SPLINE
SPL {X  -134.737, Y  +296.229, Z    +0.000, E1   +47.890, E3 +135435.927}
SPL {X  -154.917, Y  +342.531, Z    +0.000, E1   +31.203, E3 +135454.495}
SPL {X  -159.440, Y  +369.246, Z    +0.000, E1   +13.458, E3 +135458.394}
SPL {X  -159.987, Y  +381.470, Z    +0.000, E1    +2.976, E3 +135458.993}
SPL {X  -159.990, Y  +384.500, Z    +0.000, E1    +0.000, E3 +135459.026}
SPL {X  -159.990, Y  +386.323, Z    +0.000, E1    -3.079, E3 +135459.048}
SPL {X  -159.990, Y  +390.285, Z    +0.000, E1   -11.315, E3 +135459.169}
SPL {X  -159.990, Y  +394.559, Z    +0.000, E1   -20.770, E3 +135459.431}
SPL {X  -159.990, Y  +399.334, Z    +0.000, E1   -30.876, E3 +135459.870}
SPL {X  -159.990, Y  +405.006, Z    +0.000, E1   -40.810, E3 +135460.588}
SPL {X  -159.990, Y  +415.193, Z    +0.000, E1   -52.724, E3 +135462.475}
SPL {X  -159.990, Y  +465.395, Z    +0.000, E1   -68.959, E3 +135477.563}
SPL {X  -159.990, Y  +657.157, Z    +0.000, E1   -72.499, E3 +135573.960}
SPL {X  -159.693, Y  +681.249, Z    +0.000, E1   -72.488, E3 +135590.354}
SPL {X  -157.599, Y  +699.059, Z    +0.000, E1   -72.249, E3 +135604.514}
SPL {X  -155.217, Y  +710.289, Z    +0.000, E1   -71.989, E3 +135614.530}
SPL {X  -152.611, Y  +719.527, Z    +0.000, E1   -71.702, E3 +135623.352}
SPL {X  -149.536, Y  +728.383, Z    +0.000, E1   -71.359, E3 +135632.331}
SPL {X  -146.250, Y  +736.367, Z    +0.000, E1   -70.965, E3 +135640.885}
SPL {X  -143.481, Y  +742.281, Z    +0.000, E1   -70.623, E3 +135647.480}
SPL {X  -140.071, Y  +748.811, Z    +0.000, E1   -70.193, E3 +135654.992}
SPL {X  -136.578, Y  +754.826, Z    +0.000, E1   -69.723, E3 +135662.122}
SPL {X  -132.176, Y  +761.646, Z    +0.000, E1   -69.128, E3 +135670.365}
SPL {X  -127.941, Y  +767.561, Z    +0.000, E1   -68.475, E3 +135677.673}
SPL {X  -124.983, Y  +771.380, Z    +0.000, E1   -68.003, E3 +135682.392}
SPL {X  -122.624, Y  +774.263, Z    +0.000, E1   -67.622, E3 +135685.915}
SPL {X   -84.435, Y  +807.395, Z    +0.000, E1   -55.948, E3 +135796.919}
ENDSPLINE

SPLINE
SPL {X  -119.703, Y  +777.650, Z    +0.000, E1   -51.831, E3 +135960.926}
SPL {X  -145.184, Y  +738.720, Z    +0.000, E1   -43.488, E3 +135987.484}
SPL {X  -156.175, Y  +706.232, Z    +0.000, E1   -28.819, E3 +135996.369}
SPL {X  -159.337, Y  +685.942, Z    +0.000, E1   -14.672, E3 +135998.920}
SPL {X  -159.962, Y  +674.468, Z    +0.000, E1    -4.846, E3 +135999.539}
SPL {X  -159.990, Y  +669.479, Z    +0.000, E1    +0.004, E3 +135999.613}
SPL {X  -159.990, Y  +667.035, Z    +0.000, E1    +4.539, E3 +135999.644}
SPL {X  -159.990, Y  +662.914, Z    +0.000, E1   +13.494, E3 +135999.782}
SPL {X  -159.990, Y  +658.254, Z    +0.000, E1   +24.153, E3 +136000.060}
SPL {X  -159.990, Y  +650.381, Z    +0.000, E1   +39.393, E3 +136000.912}
SPL {X  -159.990, Y  +638.701, Z    +0.000, E1   +53.953, E3 +136002.798}
SPL {X  -159.990, Y  +618.566, Z    +0.000, E1   +64.119, E3 +136008.306}
SPL {X  -159.990, Y  +582.261, Z    +0.000, E1   +69.343, E3 +136021.792}
SPL {X  -159.990, Y  +406.555, Z    +0.000, E1   +71.635, E3 +136118.038}
SPL {X  -159.990, Y  +385.723, Z    +0.000, E1   +71.610, E3 +136132.777}
SPL {X  -159.404, Y  +368.814, Z    +0.000, E1   +71.556, E3 +136145.306}
SPL {X  -157.440, Y  +354.048, Z    +0.000, E1   +71.342, E3 +136157.779}
SPL {X  -155.889, Y  +346.508, Z    +0.000, E1   +70.461, E3 +136171.327}
SPL {X  -154.332, Y  +340.328, Z    +0.000, E1   +70.024, E3 +136179.555}
SPL {X  -150.579, Y  +328.438, Z    +0.000, E1   +70.374, E3 +136185.274}
SPL {X  -146.933, Y  +319.195, Z    +0.000, E1   +70.230, E3 +136192.965}
SPL {X  -143.573, Y  +311.906, Z    +0.000, E1   +69.806, E3 +136201.275}
SPL {X  -139.693, Y  +304.508, Z    +0.000, E1   +69.301, E3 +136210.003}
SPL {X  -135.622, Y  +297.627, Z    +0.000, E1   +68.731, E3 +136218.411}
SPL {X  -131.165, Y  +290.889, Z    +0.000, E1   +68.094, E3 +136226.797}
SPL {X  -126.457, Y  +284.492, Z    +0.000, E1   +67.352, E3 +136234.882}
SPL {X  -123.432, Y  +280.710, Z    +0.000, E1   +66.830, E3 +136239.668}
SPL {X   -85.607, Y  +247.340, Z    +0.000, E1   +53.917, E3 +136381.389}
ENDSPLINE

SPLINE
SPL {X  -134.737, Y  +296.229, Z    +0.000, E1   +47.890, E3 +136524.162}
SPL {X  -154.917, Y  +342.531, Z    +0.000, E1   +31.203, E3 +136542.730}
SPL {X  -159.440, Y  +369.246, Z    +0.000, E1   +13.458, E3 +136546.629}
SPL {X  -159.987, Y  +381.470, Z    +0.000, E1    +2.976, E3 +136547.228}
SPL {X  -159.990, Y  +384.500, Z    +0.000, E1    +0.000, E3 +136547.261}
SPL {X  -159.990, Y  +386.323, Z    +0.000, E1    -3.079, E3 +136547.283}
SPL {X  -159.990, Y  +390.285, Z    +0.000, E1   -11.315, E3 +136547.404}
SPL {X  -159.990, Y  +394.559, Z    +0.000, E1   -20.770, E3 +136547.666}
SPL {X  -159.990, Y  +402.118, Z    +0.000, E1   -35.793, E3 +136548.457}
SPL {X  -159.990, Y  +415.193, Z    +0.000, E1   -52.724, E3 +136550.710}
SPL {X  -159.990, Y  +465.395, Z    +0.000, E1   -68.959, E3 +136565.799}
SPL {X  -159.990, Y  +652.170, Z    +0.000, E1   -72.485, E3 +136658.894}
SPL {X  -159.990, Y  +670.864, Z    +0.000, E1   -72.509, E3 +136671.342}
SPL {X  -159.251, Y  +686.856, Z    +0.000, E1   -72.412, E3 +136682.884}
SPL {X  -157.599, Y  +699.059, Z    +0.000, E1   -72.249, E3 +136692.749}
SPL {X  -155.217, Y  +710.289, Z    +0.000, E1   -71.989, E3 +136702.766}
SPL {X  -152.611, Y  +719.527, Z    +0.000, E1   -71.702, E3 +136711.587}
SPL {X  -149.536, Y  +728.383, Z    +0.000, E1   -71.359, E3 +136720.566}
SPL {X  -146.250, Y  +736.367, Z    +0.000, E1   -70.965, E3 +136729.120}
SPL {X  -143.481, Y  +742.281, Z    +0.000, E1   -70.623, E3 +136735.716}
SPL {X  -140.071, Y  +748.811, Z    +0.000, E1   -70.193, E3 +136743.227}
SPL {X  -136.578, Y  +754.826, Z    +0.000, E1   -69.723, E3 +136750.357}
SPL {X  -133.265, Y  +760.028, Z    +0.000, E1   -69.258, E3 +136756.658}
SPL {X  -129.890, Y  +764.909, Z    +0.000, E1   -68.775, E3 +136762.628}
SPL {X  -125.802, Y  +770.346, Z    +0.000, E1   -68.156, E3 +136769.328}
SPL {X  -122.624, Y  +774.263, Z    +0.000, E1   -67.622, E3 +136774.150}
SPL {X   -84.435, Y  +807.395, Z    +0.000, E1   -55.948, E3 +136885.155}
ENDSPLINE

SPLINE
SPL {X  -119.703, Y  +777.650, Z    +0.000, E1   -51.831, E3 +137049.161}
SPL {X  -145.184, Y  +738.720, Z    +0.000, E1   -43.488, E3 +137075.719}
SPL {X  -156.175, Y  +706.232, Z    +0.000, E1   -28.819, E3 +137084.604}
SPL {X  -159.337, Y  +685.942, Z    +0.000, E1   -14.672, E3 +137087.155}
SPL {X  -159.962, Y  +674.468, Z    +0.000, E1    -4.846, E3 +137087.774}
SPL {X  -159.990, Y  +669.479, Z    +0.000, E1    +0.004, E3 +137087.848}
SPL {X  -159.990, Y  +667.035, Z    +0.000, E1    +4.539, E3 +137087.879}
SPL {X  -159.990, Y  +662.914, Z    +0.000, E1   +13.494, E3 +137088.018}
SPL {X  -159.990, Y  +658.254, Z    +0.000, E1   +24.153, E3 +137088.295}
SPL {X  -159.990, Y  +652.944, Z    +0.000, E1   +35.122, E3 +137088.799}
SPL {X  -159.990, Y  +642.509, Z    +0.000, E1   +50.090, E3 +137090.371}
SPL {X  -159.990, Y  +618.566, Z    +0.000, E1   +64.119, E3 +137096.541}
SPL {X  -159.990, Y  +584.545, Z    +0.000, E1   +69.188, E3 +137109.076}
SPL {X  -159.990, Y  +578.002, Z    +0.000, E1   +69.607, E3 +137111.800}
SPL {X  -159.990, Y  +426.570, Z    +0.000, E1   +71.599, E3 +137192.290}
SPL {X  -159.990, Y  +405.946, Z    +0.000, E1   +71.630, E3 +137206.720}
SPL {X  -159.967, Y  +379.776, Z    +0.000, E1   +71.634, E3 +137225.167}
SPL {X  -158.535, Y  +360.970, Z    +0.000, E1   +71.460, E3 +137239.989}
SPL {X  -156.277, Y  +348.230, Z    +0.000, E1   +71.211, E3 +137251.332}
SPL {X  -155.351, Y  +344.251, Z    +0.000, E1   +70.004, E3 +137265.124}
SPL {X  -150.579, Y  +328.438, Z    +0.000, E1   +70.374, E3 +137273.509}
SPL {X  -146.933, Y  +319.195, Z    +0.000, E1   +70.230, E3 +137281.200}
SPL {X  -143.573, Y  +311.906, Z    +0.000, E1   +69.806, E3 +137289.510}
SPL {X  -139.693, Y  +304.508, Z    +0.000, E1   +69.301, E3 +137298.239}
SPL {X  -135.622, Y  +297.627, Z    +0.000, E1   +68.731, E3 +137306.647}
SPL {X  -131.165, Y  +290.889, Z    +0.000, E1   +68.094, E3 +137315.032}
SPL {X  -126.457, Y  +284.492, Z    +0.000, E1   +67.352, E3 +137323.118}
SPL {X  -123.432, Y  +280.710, Z    +0.000, E1   +66.830, E3 +137327.903}
SPL {X   -85.607, Y  +247.340, Z    +0.000, E1   +53.917, E3 +137469.625}
ENDSPLINE

SPLINE
SPL {X  -134.737, Y  +296.229, Z    +0.000, E1   +47.890, E3 +137612.398}
SPL {X  -154.917, Y  +342.531, Z    +0.000, E1   +31.203, E3 +137630.965}
SPL {X  -159.440, Y  +369.246, Z    +0.000, E1   +13.458, E3 +137634.864}
SPL {X  -159.957, Y  +379.264, Z    +0.000, E1    +4.909, E3 +137635.421}
SPL {X  -159.990, Y  +384.670, Z    +0.000, E1    -0.079, E3 +137635.498}
SPL {X  -159.990, Y  +389.248, Z    +0.000, E1    -8.879, E3 +137635.602}
SPL {X  -159.990, Y  +394.559, Z    +0.000, E1   -20.770, E3 +137635.901}
SPL {X  -159.990, Y  +402.118, Z    +0.000, E1   -35.793, E3 +137636.693}
SPL {X  -159.990, Y  +415.193, Z    +0.000, E1   -52.724, E3 +137638.945}
SPL {X  -159.990, Y  +465.395, Z    +0.000, E1   -68.959, E3 +137654.034}
SPL {X  -159.990, Y  +657.157, Z    +0.000, E1   -72.499, E3 +137750.431}
SPL {X  -159.947, Y  +675.227, Z    +0.000, E1   -72.487, E3 +137762.591}
SPL {X  -159.251, Y  +686.856, Z    +0.000, E1   -72.412, E3 +137771.119}
SPL {X  -157.599, Y  +699.059, Z    +0.000, E1   -72.249, E3 +137780.984}
SPL {X  -155.217, Y  +710.289, Z    +0.000, E1   -71.989, E3 +137791.001}
SPL {X  -152.611, Y  +719.527, Z    +0.000, E1   -71.702, E3 +137799.822}
SPL {X  -149.536, Y  +728.383, Z    +0.000, E1   -71.359, E3 +137808.801}
SPL {X  -146.250, Y  +736.367, Z    +0.000, E1   -70.965, E3 +137817.356}
SPL {X  -143.481, Y  +742.281, Z    +0.000, E1   -70.623, E3 +137823.951}
SPL {X  -140.071, Y  +748.811, Z    +0.000, E1   -70.193, E3 +137831.463}
SPL {X  -136.578, Y  +754.826, Z    +0.000, E1   -69.723, E3 +137838.592}
SPL {X  -133.265, Y  +760.028, Z    +0.000, E1   -69.258, E3 +137844.893}
SPL {X  -129.890, Y  +764.909, Z    +0.000, E1   -68.775, E3 +137850.864}
SPL {X  -125.802, Y  +770.346, Z    +0.000, E1   -68.156, E3 +137857.563}
SPL {X  -122.624, Y  +774.263, Z    +0.000, E1   -67.622, E3 +137862.386}
SPL {X   -84.435, Y  +807.395, Z    +0.000, E1   -55.948, E3 +137973.390}
ENDSPLINE

SPLINE
SPL {X  -119.703, Y  +777.650, Z    +0.000, E1   -51.831, E3 +138137.397}
SPL {X  -145.184, Y  +738.720, Z    +0.000, E1   -43.488, E3 +138163.955}
SPL {X  -154.467, Y  +713.173, Z    +0.000, E1   -32.658, E3 +138171.550}
SPL {X  -157.530, Y  +699.446, Z    +0.000, E1   -24.482, E3 +138173.966}
SPL {X  -159.337, Y  +685.942, Z    +0.000, E1   -14.672, E3 +138175.391}
SPL {X  -159.962, Y  +674.468, Z    +0.000, E1    -4.846, E3 +138176.009}
SPL {X  -159.990, Y  +669.479, Z    +0.000, E1    +0.004, E3 +138176.083}
SPL {X  -159.990, Y  +667.035, Z    +0.000, E1    +4.539, E3 +138176.114}
SPL {X  -159.990, Y  +662.914, Z    +0.000, E1   +13.494, E3 +138176.253}
SPL {X  -159.990, Y  +658.254, Z    +0.000, E1   +24.153, E3 +138176.531}
SPL {X  -159.990, Y  +652.944, Z    +0.000, E1   +35.122, E3 +138177.034}
SPL {X  -159.990, Y  +642.509, Z    +0.000, E1   +50.090, E3 +138178.606}
SPL {X  -159.990, Y  +618.566, Z    +0.000, E1   +64.119, E3 +138184.777}
SPL {X  -159.990, Y  +582.261, Z    +0.000, E1   +69.343, E3 +138198.262}
SPL {X  -159.990, Y  +406.555, Z    +0.000, E1   +71.635, E3 +138294.509}
SPL {X  -159.990, Y  +385.723, Z    +0.000, E1   +71.610, E3 +138309.247}
SPL {X  -159.700, Y  +372.863, Z    +0.000, E1   +71.570, E3 +138318.653}
SPL {X  -158.535, Y  +360.970, Z    +0.000, E1   +71.460, E3 +138328.224}
SPL {X  -156.277, Y  +348.230, Z    +0.000, E1   +71.211, E3 +138339.567}
SPL {X  -155.351, Y  +344.251, Z    +0.000, E1   +70.004, E3 +138353.359}
SPL {X  -150.579, Y  +328.438, Z    +0.000, E1   +70.374, E3 +138361.744}
SPL {X  -146.933, Y  +319.195, Z    +0.000, E1   +70.230, E3 +138369.435}
SPL {X  -143.573, Y  +311.906, Z    +0.000, E1   +69.806, E3 +138377.746}
SPL {X  -140.547, Y  +306.057, Z    +0.000, E1   +69.399, E3 +138384.638}
SPL {X  -137.438, Y  +300.600, Z    +0.000, E1   +68.984, E3 +138391.232}
SPL {X  -133.397, Y  +294.172, Z    +0.000, E1   +68.416, E3 +138399.167}
SPL {X  -128.822, Y  +287.623, Z    +0.000, E1   +67.729, E3 +138407.391}
SPL {X  -124.502, Y  +282.021, Z    +0.000, E1   +67.035, E3 +138414.465}
SPL {X   -85.607, Y  +247.340, Z    +0.000, E1   +53.917, E3 +138557.860}
ENDSPLINE

SPLINE
SPL {X  -119.557, Y  +276.184, Z    +0.000, E1   +51.032, E3 +138681.397}
SPL {X  -138.294, Y  +302.054, Z    +0.000, E1   +46.576, E3 +138704.719}
SPL {X  -153.211, Y  +336.421, Z    +0.000, E1   +34.262, E3 +138717.841}
SPL {X  -158.240, Y  +358.900, Z    +0.000, E1   +21.089, E3 +138722.046}
SPL {X  -159.674, Y  +372.451, Z    +0.000, E1   +10.778, E3 +138723.342}
SPL {X  -159.987, Y  +381.470, Z    +0.000, E1    +2.976, E3 +138723.699}
SPL {X  -159.990, Y  +384.761, Z    +0.000, E1    -0.257, E3 +138723.734}
SPL {X  -159.990, Y  +389.248, Z    +0.000, E1    -8.879, E3 +138723.838}
SPL {X  -159.990, Y  +394.559, Z    +0.000, E1   -20.770, E3 +138724.137}
SPL {X  -159.990, Y  +402.118, Z    +0.000, E1   -35.793, E3 +138724.928}
SPL {X  -159.990, Y  +415.193, Z    +0.000, E1   -52.724, E3 +138727.181}
SPL {X  -159.990, Y  +465.395, Z    +0.000, E1   -68.959, E3 +138742.269}
SPL {X  -159.990, Y  +657.157, Z    +0.000, E1   -72.499, E3 +138838.666}
SPL {X  -159.693, Y  +681.249, Z    +0.000, E1   -72.488, E3 +138855.060}
SPL {X  -157.599, Y  +699.059, Z    +0.000, E1   -72.249, E3 +138869.220}
SPL {X  -155.217, Y  +710.289, Z    +0.000, E1   -71.989, E3 +138879.236}
SPL {X  -152.611, Y  +719.527, Z    +0.000, E1   -71.702, E3 +138888.058}
SPL {X  -149.536, Y  +728.383, Z    +0.000, E1   -71.359, E3 +138897.037}
SPL {X  -146.250, Y  +736.367, Z    +0.000, E1   -70.965, E3 +138905.591}
SPL {X  -143.481, Y  +742.281, Z    +0.000, E1   -70.623, E3 +138912.186}
SPL {X  -140.071, Y  +748.811, Z    +0.000, E1   -70.193, E3 +138919.698}
SPL {X  -136.578, Y  +754.826, Z    +0.000, E1   -69.723, E3 +138926.827}
SPL {X  -133.265, Y  +760.028, Z    +0.000, E1   -69.258, E3 +138933.128}
SPL {X  -129.890, Y  +764.909, Z    +0.000, E1   -68.775, E3 +138939.099}
SPL {X  -125.802, Y  +770.346, Z    +0.000, E1   -68.156, E3 +138945.798}
SPL {X  -122.624, Y  +774.263, Z    +0.000, E1   -67.622, E3 +138950.621}
SPL {X   -84.435, Y  +807.395, Z    +0.000, E1   -55.948, E3 +139061.625}
ENDSPLINE

SPLINE
SPL {X  -119.703, Y  +777.650, Z    +0.000, E1   -51.831, E3 +139225.632}
SPL {X  -145.184, Y  +738.720, Z    +0.000, E1   -43.488, E3 +139252.190}
SPL {X  -156.175, Y  +706.232, Z    +0.000, E1   -28.819, E3 +139261.075}
SPL {X  -159.337, Y  +685.942, Z    +0.000, E1   -14.672, E3 +139263.626}
SPL {X  -159.900, Y  +676.871, Z    +0.000, E1    -6.955, E3 +139264.174}
SPL {X  -159.990, Y  +669.634, Z    +0.000, E1    -0.285, E3 +139264.318}
SPL {X  -159.990, Y  +667.035, Z    +0.000, E1    +4.539, E3 +139264.349}
SPL {X  -159.990, Y  +662.914, Z    +0.000, E1   +13.494, E3 +139264.488}
SPL {X  -159.990, Y  +658.254, Z    +0.000, E1   +24.153, E3 +139264.766}
SPL {X  -159.990, Y  +652.944, Z    +0.000, E1   +35.122, E3 +139265.270}
SPL {X  -159.990, Y  +642.509, Z    +0.000, E1   +50.090, E3 +139266.841}
SPL {X  -159.990, Y  +618.566, Z    +0.000, E1   +64.119, E3 +139273.012}
SPL {X  -159.990, Y  +584.545, Z    +0.000, E1   +69.188, E3 +139285.547}
SPL {X  -159.990, Y  +578.002, Z    +0.000, E1   +69.607, E3 +139288.271}
SPL {X  -159.990, Y  +426.570, Z    +0.000, E1   +71.599, E3 +139368.761}
SPL {X  -159.990, Y  +405.946, Z    +0.000, E1   +71.630, E3 +139383.191}
SPL {X  -159.967, Y  +379.776, Z    +0.000, E1   +71.634, E3 +139401.637}
SPL {X  -158.535, Y  +360.970, Z    +0.000, E1   +71.460, E3 +139416.459}
SPL {X  -156.882, Y  +351.118, Z    +0.000, E1   +71.263, E3 +139425.171}
SPL {X  -155.538, Y  +345.018, Z    +0.000, E1   +71.109, E3 +139430.878}
SPL {X  -155.351, Y  +344.251, Z    +0.000, E1   +70.004, E3 +139441.594}
SPL {X  -150.579, Y  +328.438, Z    +0.000, E1   +70.374, E3 +139449.980}
SPL {X  -146.933, Y  +319.195, Z    +0.000, E1   +70.230, E3 +139457.671}
SPL {X  -143.573, Y  +311.906, Z    +0.000, E1   +69.806, E3 +139465.981}
SPL {X  -140.547, Y  +306.057, Z    +0.000, E1   +69.399, E3 +139472.873}
SPL {X  -137.438, Y  +300.600, Z    +0.000, E1   +68.984, E3 +139479.467}
SPL {X  -133.397, Y  +294.172, Z    +0.000, E1   +68.416, E3 +139487.402}
SPL {X  -128.822, Y  +287.623, Z    +0.000, E1   +67.729, E3 +139495.627}
SPL {X  -124.502, Y  +282.021, Z    +0.000, E1   +67.035, E3 +139502.701}
SPL {X   -85.607, Y  +247.340, Z    +0.000, E1   +53.917, E3 +139646.095}
ENDSPLINE

SPLINE
SPL {X  -134.737, Y  +296.229, Z    +0.000, E1   +47.890, E3 +139788.868}
SPL {X  -153.211, Y  +336.421, Z    +0.000, E1   +34.262, E3 +139806.076}
SPL {X  -158.240, Y  +358.900, Z    +0.000, E1   +21.089, E3 +139810.281}
SPL {X  -159.854, Y  +375.896, Z    +0.000, E1    +7.981, E3 +139811.747}
SPL {X  -159.990, Y  +384.398, Z    +0.000, E1    +0.172, E3 +139811.967}
SPL {X  -159.990, Y  +386.323, Z    +0.000, E1    -3.079, E3 +139811.989}
SPL {X  -159.990, Y  +390.285, Z    +0.000, E1   -11.315, E3 +139812.110}
SPL {X  -159.990, Y  +394.559, Z    +0.000, E1   -20.770, E3 +139812.372}
SPL {X  -159.990, Y  +399.334, Z    +0.000, E1   -30.876, E3 +139812.811}
SPL {X  -159.990, Y  +405.006, Z    +0.000, E1   -40.810, E3 +139813.529}
SPL {X  -159.990, Y  +415.193, Z    +0.000, E1   -52.724, E3 +139815.416}
SPL {X  -159.990, Y  +465.395, Z    +0.000, E1   -68.959, E3 +139830.505}
SPL {X  -159.990, Y  +657.157, Z    +0.000, E1   -72.499, E3 +139926.901}
SPL {X  -159.693, Y  +681.249, Z    +0.000, E1   -72.488, E3 +139943.295}
SPL {X  -157.599, Y  +699.059, Z    +0.000, E1   -72.249, E3 +139957.455}
SPL {X  -155.217, Y  +710.289, Z    +0.000, E1   -71.989, E3 +139967.472}
SPL {X  -152.611, Y  +719.527, Z    +0.000, E1   -71.702, E3 +139976.293}
SPL {X  -149.536, Y  +728.383, Z    +0.000, E1   -71.359, E3 +139985.272}
SPL {X  -146.250, Y  +736.367, Z    +0.000, E1   -70.965, E3 +139993.826}
SPL {X  -143.481, Y  +742.281, Z    +0.000, E1   -70.623, E3 +140000.422}
SPL {X  -140.071, Y  +748.811, Z    +0.000, E1   -70.193, E3 +140007.933}
SPL {X  -136.578, Y  +754.826, Z    +0.000, E1   -69.723, E3 +140015.063}
SPL {X  -133.265, Y  +760.028, Z    +0.000, E1   -69.258, E3 +140021.364}
SPL {X  -129.890, Y  +764.909, Z    +0.000, E1   -68.775, E3 +140027.334}
SPL {X  -125.802, Y  +770.346, Z    +0.000, E1   -68.156, E3 +140034.033}
SPL {X  -122.624, Y  +774.263, Z    +0.000, E1   -67.622, E3 +140038.856}
SPL {X   -84.435, Y  +807.395, Z    +0.000, E1   -55.948, E3 +140149.861}
ENDSPLINE

SPLINE
SPL {X  -119.703, Y  +777.650, Z    +0.000, E1   -51.831, E3 +140313.867}
SPL {X  -145.184, Y  +738.720, Z    +0.000, E1   -43.488, E3 +140340.425}
SPL {X  -156.175, Y  +706.232, Z    +0.000, E1   -28.819, E3 +140349.310}
SPL {X  -159.337, Y  +685.942, Z    +0.000, E1   -14.672, E3 +140351.861}
SPL {X  -159.900, Y  +676.871, Z    +0.000, E1    -6.955, E3 +140352.409}
SPL {X  -159.990, Y  +669.634, Z    +0.000, E1    -0.285, E3 +140352.553}
SPL {X  -159.990, Y  +667.035, Z    +0.000, E1    +4.539, E3 +140352.585}
SPL {X  -159.990, Y  +662.914, Z    +0.000, E1   +13.494, E3 +140352.724}
SPL {X  -159.990, Y  +658.254, Z    +0.000, E1   +24.153, E3 +140353.001}
SPL {X  -159.990, Y  +652.944, Z    +0.000, E1   +35.122, E3 +140353.505}
SPL {X  -159.990, Y  +646.557, Z    +0.000, E1   +45.390, E3 +140354.372}
SPL {X  -159.990, Y  +638.701, Z    +0.000, E1   +53.953, E3 +140355.739}
SPL {X  -159.990, Y  +618.566, Z    +0.000, E1   +64.119, E3 +140361.247}
SPL {X  -159.990, Y  +582.261, Z    +0.000, E1   +69.343, E3 +140374.733}
SPL {X  -159.990, Y  +414.423, Z    +0.000, E1   +71.602, E3 +140465.516}
SPL {X  -159.990, Y  +400.357, Z    +0.000, E1   +71.604, E3 +140475.427}
SPL {X  -159.990, Y  +385.723, Z    +0.000, E1   +71.610, E3 +140485.718}
SPL {X  -159.404, Y  +368.814, Z    +0.000, E1   +71.556, E3 +140498.247}
SPL {X  -157.440, Y  +354.048, Z    +0.000, E1   +71.342, E3 +140510.720}
SPL {X  -155.889, Y  +346.508, Z    +0.000, E1   +70.461, E3 +140524.268}
SPL {X  -154.332, Y  +340.328, Z    +0.000, E1   +70.024, E3 +140532.496}
SPL {X  -150.579, Y  +328.438, Z    +0.000, E1   +70.374, E3 +140538.215}
SPL {X  -146.933, Y  +319.195, Z    +0.000, E1   +70.230, E3 +140545.906}
SPL {X  -143.573, Y  +311.906, Z    +0.000, E1   +69.806, E3 +140554.216}
SPL {X  -139.693, Y  +304.508, Z    +0.000, E1   +69.301, E3 +140562.945}
SPL {X  -135.622, Y  +297.627, Z    +0.000, E1   +68.731, E3 +140571.353}
SPL {X  -132.531, Y  +292.877, Z    +0.000, E1   +68.266, E3 +140577.288}
SPL {X  -128.822, Y  +287.623, Z    +0.000, E1   +67.729, E3 +140583.862}
SPL {X  -124.502, Y  +282.021, Z    +0.000, E1   +67.035, E3 +140590.936}
SPL {X   -85.607, Y  +247.340, Z    +0.000, E1   +53.917, E3 +140734.331}
ENDSPLINE

SPLINE
SPL {X  -134.737, Y  +296.229, Z    +0.000, E1   +47.890, E3 +140877.103}
SPL {X  -154.917, Y  +342.531, Z    +0.000, E1   +31.203, E3 +140895.671}
SPL {X  -159.440, Y  +369.246, Z    +0.000, E1   +13.458, E3 +140899.570}
SPL {X  -159.987, Y  +381.470, Z    +0.000, E1    +2.976, E3 +140900.169}
SPL {X  -159.990, Y  +384.500, Z    +0.000, E1    +0.000, E3 +140900.203}
SPL {X  -159.990, Y  +386.323, Z    +0.000, E1    -3.079, E3 +140900.224}
SPL {X  -159.990, Y  +390.285, Z    +0.000, E1   -11.315, E3 +140900.345}
SPL {X  -159.990, Y  +394.559, Z    +0.000, E1   -20.770, E3 +140900.607}
SPL {X  -159.990, Y  +402.118, Z    +0.000, E1   -35.793, E3 +140901.399}
SPL {X  -159.990, Y  +415.193, Z    +0.000, E1   -52.724, E3 +140903.651}
SPL {X  -159.990, Y  +465.395, Z    +0.000, E1   -68.959, E3 +140918.740}
SPL {X  -159.990, Y  +657.157, Z    +0.000, E1   -72.499, E3 +141015.137}
SPL {X  -159.693, Y  +681.249, Z    +0.000, E1   -72.488, E3 +141031.531}
SPL {X  -157.599, Y  +699.059, Z    +0.000, E1   -72.249, E3 +141045.690}
SPL {X  -155.217, Y  +710.289, Z    +0.000, E1   -71.989, E3 +141055.707}
SPL {X  -152.611, Y  +719.527, Z    +0.000, E1   -71.702, E3 +141064.528}
SPL {X  -149.536, Y  +728.383, Z    +0.000, E1   -71.359, E3 +141073.507}
SPL {X  -146.250, Y  +736.367, Z    +0.000, E1   -70.965, E3 +141082.061}
SPL {X  -143.481, Y  +742.281, Z    +0.000, E1   -70.623, E3 +141088.657}
SPL {X  -140.071, Y  +748.811, Z    +0.000, E1   -70.193, E3 +141096.169}
SPL {X  -136.578, Y  +754.826, Z    +0.000, E1   -69.723, E3 +141103.298}
SPL {X  -133.265, Y  +760.028, Z    +0.000, E1   -69.258, E3 +141109.599}
SPL {X  -129.890, Y  +764.909, Z    +0.000, E1   -68.775, E3 +141115.570}
SPL {X  -125.802, Y  +770.346, Z    +0.000, E1   -68.156, E3 +141122.269}
SPL {X  -122.624, Y  +774.263, Z    +0.000, E1   -67.622, E3 +141127.091}
SPL {X   -84.435, Y  +807.395, Z    +0.000, E1   -55.948, E3 +141238.096}
ENDSPLINE

SPLINE
SPL {X  -119.703, Y  +777.650, Z    +0.000, E1   -51.831, E3 +141402.103}
SPL {X  -145.184, Y  +738.720, Z    +0.000, E1   -43.488, E3 +141428.661}
SPL {X  -156.175, Y  +706.232, Z    +0.000, E1   -28.819, E3 +141437.545}
SPL {X  -159.337, Y  +685.942, Z    +0.000, E1   -14.672, E3 +141440.097}
SPL {X  -159.962, Y  +674.468, Z    +0.000, E1    -4.846, E3 +141440.715}
SPL {X  -159.990, Y  +669.479, Z    +0.000, E1    +0.004, E3 +141440.789}
SPL {X  -159.990, Y  +667.035, Z    +0.000, E1    +4.539, E3 +141440.820}
SPL {X  -159.990, Y  +662.914, Z    +0.000, E1   +13.494, E3 +141440.959}
SPL {X  -159.990, Y  +658.254, Z    +0.000, E1   +24.153, E3 +141441.237}
SPL {X  -159.990, Y  +652.944, Z    +0.000, E1   +35.122, E3 +141441.740}
SPL {X  -159.990, Y  +642.509, Z    +0.000, E1   +50.090, E3 +141443.312}
SPL {X  -159.990, Y  +618.566, Z    +0.000, E1   +64.119, E3 +141449.482}
SPL {X  -159.990, Y  +584.545, Z    +0.000, E1   +69.188, E3 +141462.018}
SPL {X  -159.990, Y  +578.002, Z    +0.000, E1   +69.607, E3 +141464.741}
SPL {X  -159.990, Y  +426.570, Z    +0.000, E1   +71.599, E3 +141545.231}
SPL {X  -159.990, Y  +405.946, Z    +0.000, E1   +71.630, E3 +141559.661}
SPL {X  -159.967, Y  +379.776, Z    +0.000, E1   +71.634, E3 +141578.108}
SPL {X  -158.535, Y  +360.970, Z    +0.000, E1   +71.460, E3 +141592.930}
SPL {X  -156.277, Y  +348.230, Z    +0.000, E1   +71.211, E3 +141604.273}
SPL {X  -155.351, Y  +344.251, Z    +0.000, E1   +70.004, E3 +141618.065}
SPL {X  -150.579, Y  +328.438, Z    +0.000, E1   +70.374, E3 +141626.450}
SPL {X  -146.933, Y  +319.195, Z    +0.000, E1   +70.230, E3 +141634.141}
SPL {X  -143.573, Y  +311.906, Z    +0.000, E1   +69.806, E3 +141642.452}
SPL {X  -139.693, Y  +304.508, Z    +0.000, E1   +69.301, E3 +141651.180}
SPL {X  -135.622, Y  +297.627, Z    +0.000, E1   +68.731, E3 +141659.588}
SPL {X  -131.165, Y  +290.889, Z    +0.000, E1   +68.094, E3 +141667.973}
SPL {X  -126.457, Y  +284.492, Z    +0.000, E1   +67.352, E3 +141676.059}
SPL {X  -123.432, Y  +280.710, Z    +0.000, E1   +66.830, E3 +141680.845}
SPL {X   -85.607, Y  +247.340, Z    +0.000, E1   +53.917, E3 +141822.566}
ENDSPLINE

SPLINE
SPL {X  -134.737, Y  +296.229, Z    +0.000, E1   +47.890, E3 +141965.339}
SPL {X  -154.917, Y  +342.531, Z    +0.000, E1   +31.203, E3 +141983.906}
SPL {X  -159.440, Y  +369.246, Z    +0.000, E1   +13.458, E3 +141987.806}
SPL {X  -159.987, Y  +381.470, Z    +0.000, E1    +2.976, E3 +141988.405}
SPL {X  -159.990, Y  +384.500, Z    +0.000, E1    +0.000, E3 +141988.438}
SPL {X  -159.990, Y  +386.323, Z    +0.000, E1    -3.079, E3 +141988.459}
SPL {X  -159.990, Y  +390.285, Z    +0.000, E1   -11.315, E3 +141988.580}
SPL {X  -159.990, Y  +394.559, Z    +0.000, E1   -20.770, E3 +141988.843}
SPL {X  -159.990, Y  +402.118, Z    +0.000, E1   -35.793, E3 +141989.634}
SPL {X  -159.990, Y  +415.193, Z    +0.000, E1   -52.724, E3 +141991.886}
SPL {X  -159.990, Y  +465.395, Z    +0.000, E1   -68.959, E3 +142006.975}
SPL {X  -159.990, Y  +657.157, Z    +0.000, E1   -72.499, E3 +142103.372}
SPL {X  -159.693, Y  +681.249, Z    +0.000, E1   -72.488, E3 +142119.766}
SPL {X  -157.599, Y  +699.059, Z    +0.000, E1   -72.249, E3 +142133.926}
SPL {X  -155.217, Y  +710.289, Z    +0.000, E1   -71.989, E3 +142143.942}
SPL {X  -152.611, Y  +719.527, Z    +0.000, E1   -71.702, E3 +142152.763}
SPL {X  -149.536, Y  +728.383, Z    +0.000, E1   -71.359, E3 +142161.743}
SPL {X  -146.250, Y  +736.367, Z    +0.000, E1   -70.965, E3 +142170.297}
SPL {X  -143.481, Y  +742.281, Z    +0.000, E1   -70.623, E3 +142176.892}
SPL {X  -140.071, Y  +748.811, Z    +0.000, E1   -70.193, E3 +142184.404}
SPL {X  -136.578, Y  +754.826, Z    +0.000, E1   -69.723, E3 +142191.533}
SPL {X  -133.265, Y  +760.028, Z    +0.000, E1   -69.258, E3 +142197.834}
SPL {X  -129.890, Y  +764.909, Z    +0.000, E1   -68.775, E3 +142203.805}
SPL {X  -125.802, Y  +770.346, Z    +0.000, E1   -68.156, E3 +142210.504}
SPL {X  -122.624, Y  +774.263, Z    +0.000, E1   -67.622, E3 +142215.327}
SPL {X   -84.435, Y  +807.395, Z    +0.000, E1   -55.948, E3 +142326.331}
ENDSPLINE

SPLINE
SPL {X  -119.703, Y  +777.650, Z    +0.000, E1   -51.831, E3 +142490.338}
SPL {X  -145.184, Y  +738.720, Z    +0.000, E1   -43.488, E3 +142516.896}
SPL {X  -156.175, Y  +706.232, Z    +0.000, E1   -28.819, E3 +142525.781}
SPL {X  -159.337, Y  +685.942, Z    +0.000, E1   -14.672, E3 +142528.332}
SPL {X  -159.962, Y  +674.468, Z    +0.000, E1    -4.846, E3 +142528.950}
SPL {X  -159.990, Y  +669.479, Z    +0.000, E1    +0.004, E3 +142529.025}
SPL {X  -159.990, Y  +667.035, Z    +0.000, E1    +4.539, E3 +142529.055}
SPL {X  -159.990, Y  +662.914, Z    +0.000, E1   +13.494, E3 +142529.194}
SPL {X  -159.990, Y  +658.254, Z    +0.000, E1   +24.153, E3 +142529.472}
SPL {X  -159.990, Y  +652.944, Z    +0.000, E1   +35.122, E3 +142529.976}
SPL {X  -159.990, Y  +642.509, Z    +0.000, E1   +50.090, E3 +142531.547}
SPL {X  -159.990, Y  +618.566, Z    +0.000, E1   +64.119, E3 +142537.718}
SPL {X  -159.990, Y  +584.545, Z    +0.000, E1   +69.188, E3 +142550.253}
SPL {X  -159.990, Y  +578.002, Z    +0.000, E1   +69.607, E3 +142552.977}
SPL {X  -159.990, Y  +426.570, Z    +0.000, E1   +71.599, E3 +142633.467}
SPL {X  -159.990, Y  +405.946, Z    +0.000, E1   +71.630, E3 +142647.897}
SPL {X  -159.967, Y  +379.776, Z    +0.000, E1   +71.634, E3 +142666.343}
SPL {X  -158.535, Y  +360.970, Z    +0.000, E1   +71.460, E3 +142681.165}
SPL {X  -156.277, Y  +348.230, Z    +0.000, E1   +71.211, E3 +142692.508}
SPL {X  -155.351, Y  +344.251, Z    +0.000, E1   +70.004, E3 +142706.300}
SPL {X  -150.579, Y  +328.438, Z    +0.000, E1   +70.374, E3 +142714.686}
ENDSPLINE

SPLINE
SPL {X  -151.964, Y  +332.463, Z    +0.000, E1   +68.042, E3 +142730.481}
ENDSPLINE

SPLINE
SPL {X  -148.519, Y  +323.011, Z    +0.000, E1   +67.572, E3 +142741.612}
SPL {X  -144.736, Y  +314.321, Z    +0.000, E1   +67.058, E3 +142752.309}
SPL {X  -140.646, Y  +306.241, Z    +0.000, E1   +66.458, E3 +142762.688}
SPL {X  -136.388, Y  +298.863, Z    +0.000, E1   +65.814, E3 +142772.461}
SPL {X  -132.805, Y  +293.283, Z    +0.000, E1   +65.214, E3 +142780.050}
SPL {X  -130.038, Y  +289.296, Z    +0.000, E1   +64.749, E3 +142785.524}
SPL {X  -127.114, Y  +285.347, Z    +0.000, E1   +64.250, E3 +142790.947}
SPL {X   -96.237, Y  +254.690, Z    +0.000, E1   +52.223, E3 +142934.335}
ENDSPLINE

SPLINE
SPL {X  -139.640, Y  +304.414, Z    +0.000, E1   +43.367, E3 +143054.696}
SPL {X  -154.086, Y  +339.440, Z    +0.000, E1   +30.439, E3 +143070.253}
SPL {X  -158.589, Y  +361.372, Z    +0.000, E1   +17.765, E3 +143074.633}
SPL {X  -159.702, Y  +372.901, Z    +0.000, E1    +9.563, E3 +143075.865}
SPL {X  -159.980, Y  +380.731, Z    +0.000, E1    +3.359, E3 +143076.263}
SPL {X  -159.990, Y  +384.465, Z    +0.000, E1    +0.049, E3 +143076.320}
SPL {X  -159.990, Y  +386.161, Z    +0.000, E1    -2.359, E3 +143076.343}
SPL {X  -159.990, Y  +390.716, Z    +0.000, E1   -10.524, E3 +143076.518}
SPL {X  -159.990, Y  +397.792, Z    +0.000, E1   -24.215, E3 +143077.148}
SPL {X  -159.990, Y  +406.707, Z    +0.000, E1   -39.277, E3 +143078.489}
SPL {X  -159.990, Y  +418.467, Z    +0.000, E1   -51.591, E3 +143081.095}
SPL {X  -159.990, Y  +469.047, Z    +0.000, E1   -66.225, E3 +143100.172}
SPL {X  -159.990, Y  +610.501, Z    +0.000, E1   -69.067, E3 +143187.776}
SPL {X  -159.990, Y  +630.690, Z    +0.000, E1   -69.080, E3 +143204.156}
SPL {X  -159.990, Y  +652.219, Z    +0.000, E1   -69.078, E3 +143221.640}
SPL {X  -159.990, Y  +671.254, Z    +0.000, E1   -69.063, E3 +143237.141}
SPL {X  -159.172, Y  +687.655, Z    +0.000, E1   -68.973, E3 +143251.301}
SPL {X  -157.106, Y  +701.739, Z    +0.000, E1   -68.720, E3 +143264.909}
SPL {X  -154.598, Y  +712.687, Z    +0.000, E1   -68.393, E3 +143276.424}
SPL {X  -151.859, Y  +721.854, Z    +0.000, E1   -68.046, E3 +143286.643}
SPL {X  -148.628, Y  +730.715, Z    +0.000, E1   -67.614, E3 +143297.052}
SPL {X  -145.416, Y  +738.215, Z    +0.000, E1   -67.166, E3 +143306.260}
SPL {X  -142.090, Y  +745.034, Z    +0.000, E1   -66.692, E3 +143314.916}
SPL {X  -138.343, Y  +751.861, Z    +0.000, E1   -66.137, E3 +143323.843}
SPL {X  -134.819, Y  +757.643, Z    +0.000, E1   -65.575, E3 +143331.609}
SPL {X  -131.187, Y  +763.079, Z    +0.000, E1   -64.994, E3 +143338.992}
SPL {X  -127.405, Y  +768.272, Z    +0.000, E1   -64.349, E3 +143346.113}
SPL {X   -94.830, Y  +800.357, Z    +0.000, E1   -53.815, E3 +143460.645}
ENDSPLINE

SPLINE
SPL {X  -133.930, Y  +759.019, Z    +0.000, E1   -46.142, E3 +143608.028}
SPL {X  -149.331, Y  +728.920, Z    +0.000, E1   -37.154, E3 +143625.199}
SPL {X  -155.856, Y  +707.636, Z    +0.000, E1   -27.210, E3 +143631.202}
SPL {X  -159.260, Y  +686.764, Z    +0.000, E1   -14.026, E3 +143634.477}
SPL {X  -159.985, Y  +672.780, Z    +0.000, E1    -3.059, E3 +143635.378}
SPL {X  -159.990, Y  +669.259, Z    +0.000, E1    +0.225, E3 +143635.433}
SPL {X  -159.990, Y  +665.054, Z    +0.000, E1    +7.292, E3 +143635.538}
SPL {X  -159.990, Y  +658.864, Z    +0.000, E1   +19.708, E3 +143635.927}
SPL {X  -159.990, Y  +650.462, Z    +0.000, E1   +35.240, E3 +143636.938}
SPL {X  -159.990, Y  +636.155, Z    +0.000, E1   +51.890, E3 +143639.835}
SPL {X  -159.990, Y  +583.574, Z    +0.000, E1   +66.740, E3 +143659.631}
SPL {X  -159.990, Y  +451.342, Z    +0.000, E1   +68.591, E3 +143745.323}
ENDSPLINE

SPLINE
SPL {X  -159.990, Y  +495.016, Z    +0.000, E1   +61.398, E3 +143759.288}
ENDSPLINE

SPLINE
SPL {X  -159.990, Y  +469.556, Z    +0.000, E1   +62.943, E3 +143776.727}
SPL {X  -159.990, Y  +452.168, Z    +0.000, E1   +63.738, E3 +143789.283}
SPL {X  -159.990, Y  +433.781, Z    +0.000, E1   +64.535, E3 +143802.308}
SPL {X  -159.990, Y  +414.623, Z    +0.000, E1   +65.374, E3 +143814.728}
SPL {X  -159.990, Y  +395.826, Z    +0.000, E1   +66.138, E3 +143826.742}
SPL {X  -159.536, Y  +370.459, Z    +0.000, E1   +67.052, E3 +143842.635}
SPL {X  -157.113, Y  +352.293, Z    +0.000, E1   +67.811, E3 +143852.217}
SPL {X  -153.587, Y  +337.689, Z    +0.000, E1   +68.173, E3 +143861.581}
SPL {X  -150.185, Y  +327.353, Z    +0.000, E1   +67.790, E3 +143872.813}
SPL {X  -147.824, Y  +321.305, Z    +0.000, E1   +67.459, E3 +143880.076}
SPL {X  -144.736, Y  +314.321, Z    +0.000, E1   +67.058, E3 +143888.673}
SPL {X  -141.667, Y  +308.155, Z    +0.000, E1   +66.586, E3 +143896.594}
SPL {X  -138.502, Y  +302.413, Z    +0.000, E1   +66.138, E3 +143904.090}
SPL {X  -135.296, Y  +297.108, Z    +0.000, E1   +65.610, E3 +143911.230}
SPL {X  -132.805, Y  +293.283, Z    +0.000, E1   +65.214, E3 +143916.413}
SPL {X  -130.038, Y  +289.296, Z    +0.000, E1   +64.749, E3 +143921.888}
SPL {X  -127.114, Y  +285.347, Z    +0.000, E1   +64.250, E3 +143927.311}
SPL {X   -96.237, Y  +254.690, Z    +0.000, E1   +52.223, E3 +144070.699}
ENDSPLINE

SPLINE
SPL {X  -139.640, Y  +304.414, Z    +0.000, E1   +43.367, E3 +144191.060}
SPL {X  -154.086, Y  +339.440, Z    +0.000, E1   +30.439, E3 +144206.617}
SPL {X  -158.589, Y  +361.372, Z    +0.000, E1   +17.765, E3 +144210.997}
SPL {X  -159.702, Y  +372.901, Z    +0.000, E1    +9.563, E3 +144212.229}
SPL {X  -159.980, Y  +380.731, Z    +0.000, E1    +3.359, E3 +144212.627}
SPL {X  -159.990, Y  +384.465, Z    +0.000, E1    +0.049, E3 +144212.684}
SPL {X  -159.990, Y  +385.295, Z    +0.000, E1    -1.130, E3 +144212.690}
SPL {X  -159.990, Y  +387.941, Z    +0.000, E1    -5.453, E3 +144212.753}
SPL {X  -159.990, Y  +392.683, Z    +0.000, E1   -14.335, E3 +144213.011}
SPL {X  -159.990, Y  +399.462, Z    +0.000, E1   -27.551, E3 +144213.697}
SPL {X  -159.990, Y  +406.707, Z    +0.000, E1   -39.277, E3 +144214.853}
SPL {X  -159.990, Y  +418.467, Z    +0.000, E1   -51.591, E3 +144217.458}
SPL {X  -159.990, Y  +469.047, Z    +0.000, E1   -66.225, E3 +144236.535}
SPL {X  -159.990, Y  +610.501, Z    +0.000, E1   -69.067, E3 +144324.139}
SPL {X  -159.990, Y  +623.913, Z    +0.000, E1   -69.046, E3 +144335.088}
SPL {X  -159.990, Y  +635.131, Z    +0.000, E1   -69.053, E3 +144344.189}
SPL {X  -159.990, Y  +648.088, Z    +0.000, E1   -69.056, E3 +144354.696}
SPL {X  -159.990, Y  +667.800, Z    +0.000, E1   -69.089, E3 +144370.645}
SPL {X  -159.471, Y  +684.377, Z    +0.000, E1   -68.989, E3 +144384.732}
SPL {X  -158.115, Y  +695.924, Z    +0.000, E1   -68.836, E3 +144395.516}
SPL {X  -156.463, Y  +704.909, Z    +0.000, E1   -68.615, E3 +144404.573}
SPL {X  -153.837, Y  +715.444, Z    +0.000, E1   -68.325, E3 +144415.750}
SPL {X  -151.088, Y  +724.124, Z    +0.000, E1   -67.925, E3 +144425.661}
SPL {X  -148.628, Y  +730.715, Z    +0.000, E1   -67.614, E3 +144433.415}
SPL {X  -145.416, Y  +738.215, Z    +0.000, E1   -67.166, E3 +144442.624}
SPL {X  -142.090, Y  +745.034, Z    +0.000, E1   -66.692, E3 +144451.279}
SPL {X  -138.343, Y  +751.861, Z    +0.000, E1   -66.137, E3 +144460.206}
SPL {X  -133.893, Y  +759.076, Z    +0.000, E1   -65.453, E3 +144469.882}
SPL {X  -130.341, Y  +764.280, Z    +0.000, E1   -64.831, E3 +144477.021}
SPL {X  -127.405, Y  +768.272, Z    +0.000, E1   -64.349, E3 +144482.476}
SPL {X   -94.830, Y  +800.357, Z    +0.000, E1   -53.815, E3 +144597.008}
ENDSPLINE

SPLINE
SPL {X  -133.930, Y  +759.019, Z    +0.000, E1   -46.142, E3 +144744.392}
SPL {X  -149.331, Y  +728.920, Z    +0.000, E1   -37.154, E3 +144761.562}
SPL {X  -155.856, Y  +707.636, Z    +0.000, E1   -27.210, E3 +144767.566}
SPL {X  -158.677, Y  +691.955, Z    +0.000, E1   -17.570, E3 +144770.271}
SPL {X  -159.802, Y  +679.261, Z    +0.000, E1    -8.330, E3 +144771.468}
SPL {X  -159.990, Y  +669.767, Z    +0.000, E1    -0.394, E3 +144771.793}
SPL {X  -159.990, Y  +667.882, Z    +0.000, E1    +2.380, E3 +144771.815}
SPL {X  -159.990, Y  +664.041, Z    +0.000, E1    +9.423, E3 +144771.941}
SPL {X  -159.990, Y  +660.147, Z    +0.000, E1   +17.275, E3 +144772.178}
SPL {X  -159.990, Y  +656.649, Z    +0.000, E1   +24.355, E3 +144772.484}
SPL {X  -159.990, Y  +650.462, Z    +0.000, E1   +35.240, E3 +144773.301}
SPL {X  -159.990, Y  +636.155, Z    +0.000, E1   +51.890, E3 +144776.199}
SPL {X  -159.990, Y  +583.574, Z    +0.000, E1   +66.740, E3 +144795.995}
SPL {X  -159.990, Y  +451.342, Z    +0.000, E1   +68.591, E3 +144881.687}
ENDSPLINE

SPLINE
SPL {X  -159.990, Y  +495.016, Z    +0.000, E1   +61.398, E3 +144895.651}
ENDSPLINE

SPLINE
SPL {X  -159.990, Y  +469.556, Z    +0.000, E1   +62.943, E3 +144913.091}
SPL {X  -159.990, Y  +445.297, Z    +0.000, E1   +64.051, E3 +144930.580}
SPL {X  -159.990, Y  +420.812, Z    +0.000, E1   +65.111, E3 +144947.171}
SPL {X  -159.990, Y  +395.826, Z    +0.000, E1   +66.138, E3 +144963.106}
SPL {X  -159.536, Y  +370.459, Z    +0.000, E1   +67.052, E3 +144978.999}
SPL {X  -155.924, Y  +346.662, Z    +0.000, E1   +68.026, E3 +144991.624}
SPL {X  -152.004, Y  +332.585, Z    +0.000, E1   +68.049, E3 +145003.062}
SPL {X  -148.519, Y  +323.011, Z    +0.000, E1   +67.572, E3 +145014.339}
SPL {X  -144.736, Y  +314.321, Z    +0.000, E1   +67.058, E3 +145025.036}
SPL {X  -140.646, Y  +306.241, Z    +0.000, E1   +66.458, E3 +145035.415}
SPL {X  -136.388, Y  +298.863, Z    +0.000, E1   +65.814, E3 +145045.188}
SPL {X  -132.805, Y  +293.283, Z    +0.000, E1   +65.214, E3 +145052.777}
SPL {X  -130.038, Y  +289.296, Z    +0.000, E1   +64.749, E3 +145058.251}
SPL {X  -127.114, Y  +285.347, Z    +0.000, E1   +64.250, E3 +145063.674}
SPL {X   -96.237, Y  +254.690, Z    +0.000, E1   +52.223, E3 +145207.062}
ENDSPLINE

SPLINE
SPL {X  -139.640, Y  +304.414, Z    +0.000, E1   +43.367, E3 +145327.423}
SPL {X  -154.086, Y  +339.440, Z    +0.000, E1   +30.439, E3 +145342.981}
SPL {X  -158.589, Y  +361.372, Z    +0.000, E1   +17.765, E3 +145347.360}
SPL {X  -159.702, Y  +372.901, Z    +0.000, E1    +9.563, E3 +145348.592}
SPL {X  -159.980, Y  +380.731, Z    +0.000, E1    +3.359, E3 +145348.990}
SPL {X  -159.990, Y  +384.465, Z    +0.000, E1    +0.049, E3 +145349.048}
SPL {X  -159.990, Y  +386.161, Z    +0.000, E1    -2.359, E3 +145349.070}
SPL {X  -159.990, Y  +390.716, Z    +0.000, E1   -10.524, E3 +145349.245}
SPL {X  -159.990, Y  +397.792, Z    +0.000, E1   -24.215, E3 +145349.875}
SPL {X  -159.990, Y  +406.707, Z    +0.000, E1   -39.277, E3 +145351.216}
SPL {X  -159.990, Y  +418.467, Z    +0.000, E1   -51.591, E3 +145353.822}
SPL {X  -159.990, Y  +469.047, Z    +0.000, E1   -66.225, E3 +145372.899}
SPL {X  -159.990, Y  +610.501, Z    +0.000, E1   -69.067, E3 +145460.503}
SPL {X  -159.990, Y  +623.913, Z    +0.000, E1   -69.046, E3 +145471.452}
SPL {X  -159.990, Y  +635.131, Z    +0.000, E1   -69.053, E3 +145480.552}
SPL {X  -159.990, Y  +648.088, Z    +0.000, E1   -69.056, E3 +145491.060}
SPL {X  -159.990, Y  +667.800, Z    +0.000, E1   -69.089, E3 +145507.008}
SPL {X  -159.172, Y  +687.655, Z    +0.000, E1   -68.973, E3 +145524.028}
SPL {X  -157.106, Y  +701.739, Z    +0.000, E1   -68.720, E3 +145537.636}
SPL {X  -153.837, Y  +715.444, Z    +0.000, E1   -68.325, E3 +145552.114}
SPL {X  -151.088, Y  +724.124, Z    +0.000, E1   -67.925, E3 +145562.024}
SPL {X  -148.628, Y  +730.715, Z    +0.000, E1   -67.614, E3 +145569.779}
SPL {X  -145.416, Y  +738.215, Z    +0.000, E1   -67.166, E3 +145578.988}
SPL {X  -142.090, Y  +745.034, Z    +0.000, E1   -66.692, E3 +145587.643}
SPL {X  -138.343, Y  +751.861, Z    +0.000, E1   -66.137, E3 +145596.570}
SPL {X  -133.893, Y  +759.076, Z    +0.000, E1   -65.453, E3 +145606.246}
SPL {X  -130.341, Y  +764.280, Z    +0.000, E1   -64.831, E3 +145613.384}
SPL {X  -127.405, Y  +768.272, Z    +0.000, E1   -64.349, E3 +145618.840}
SPL {X   -94.830, Y  +800.357, Z    +0.000, E1   -53.815, E3 +145733.372}
ENDSPLINE

SPLINE
SPL {X  -133.930, Y  +759.019, Z    +0.000, E1   -46.142, E3 +145880.755}
SPL {X  -149.331, Y  +728.920, Z    +0.000, E1   -37.154, E3 +145897.926}
SPL {X  -155.856, Y  +707.636, Z    +0.000, E1   -27.210, E3 +145903.929}
SPL {X  -159.260, Y  +686.764, Z    +0.000, E1   -14.026, E3 +145907.204}
SPL {X  -159.985, Y  +672.780, Z    +0.000, E1    -3.059, E3 +145908.105}
SPL {X  -159.990, Y  +669.500, Z    +0.000, E1    +0.000, E3 +145908.159}
SPL {X  -159.990, Y  +667.882, Z    +0.000, E1    +2.380, E3 +145908.178}
SPL {X  -159.990, Y  +664.041, Z    +0.000, E1    +9.423, E3 +145908.304}
SPL {X  -159.990, Y  +660.147, Z    +0.000, E1   +17.275, E3 +145908.541}
SPL {X  -159.990, Y  +656.649, Z    +0.000, E1   +24.355, E3 +145908.848}
SPL {X  -159.990, Y  +650.462, Z    +0.000, E1   +35.240, E3 +145909.665}
SPL {X  -159.990, Y  +636.155, Z    +0.000, E1   +51.890, E3 +145912.563}
SPL {X  -159.990, Y  +583.574, Z    +0.000, E1   +66.740, E3 +145932.359}
SPL {X  -159.990, Y  +451.342, Z    +0.000, E1   +68.591, E3 +146018.051}
ENDSPLINE

SPLINE
SPL {X  -159.990, Y  +495.016, Z    +0.000, E1   +61.398, E3 +146032.015}
ENDSPLINE

SPLINE
SPL {X  -159.990, Y  +473.575, Z    +0.000, E1   +62.704, E3 +146046.750}
SPL {X  -159.990, Y  +455.620, Z    +0.000, E1   +63.615, E3 +146059.368}
SPL {X  -159.990, Y  +439.579, Z    +0.000, E1   +64.263, E3 +146071.103}
SPL {X  -159.990, Y  +420.812, Z    +0.000, E1   +65.111, E3 +146083.535}
SPL {X  -159.990, Y  +400.802, Z    +0.000, E1   +65.940, E3 +146096.276}
SPL {X  -159.990, Y  +383.383, Z    +0.000, E1   +66.590, E3 +146107.373}
SPL {X  -158.268, Y  +359.089, Z    +0.000, E1   +67.514, E3 +146121.574}
SPL {X  -153.587, Y  +337.689, Z    +0.000, E1   +68.173, E3 +146134.308}
SPL {X  -150.185, Y  +327.353, Z    +0.000, E1   +67.790, E3 +146145.540}
SPL {X  -147.824, Y  +321.305, Z    +0.000, E1   +67.459, E3 +146152.804}
SPL {X  -144.736, Y  +314.321, Z    +0.000, E1   +67.058, E3 +146161.400}
SPL {X  -140.646, Y  +306.241, Z    +0.000, E1   +66.458, E3 +146171.779}
SPL {X  -137.570, Y  +300.823, Z    +0.000, E1   +65.968, E3 +146178.970}
SPL {X  -133.815, Y  +294.806, Z    +0.000, E1   +65.413, E3 +146187.023}
SPL {X  -130.038, Y  +289.296, Z    +0.000, E1   +64.749, E3 +146194.615}
SPL {X  -127.114, Y  +285.347, Z    +0.000, E1   +64.250, E3 +146200.038}
SPL {X   -96.237, Y  +254.690, Z    +0.000, E1   +52.223, E3 +146343.426}
ENDSPLINE

SPLINE
SPL {X  -139.640, Y  +304.414, Z    +0.000, E1   +43.367, E3 +146463.787}
SPL {X  -154.086, Y  +339.440, Z    +0.000, E1   +30.439, E3 +146479.344}
SPL {X  -158.589, Y  +361.372, Z    +0.000, E1   +17.765, E3 +146483.724}
SPL {X  -159.702, Y  +372.901, Z    +0.000, E1    +9.563, E3 +146484.956}
SPL {X  -159.980, Y  +380.731, Z    +0.000, E1    +3.359, E3 +146485.354}
SPL {X  -159.990, Y  +384.465, Z    +0.000, E1    +0.049, E3 +146485.411}
SPL {X  -159.990, Y  +386.161, Z    +0.000, E1    -2.359, E3 +146485.434}
SPL {X  -159.990, Y  +391.786, Z    +0.000, E1   -12.382, E3 +146485.685}
SPL {X  -159.990, Y  +399.462, Z    +0.000, E1   -27.551, E3 +146486.424}
SPL {X  -159.990, Y  +406.707, Z    +0.000, E1   -39.277, E3 +146487.580}
SPL {X  -159.990, Y  +418.467, Z    +0.000, E1   -51.591, E3 +146490.185}
SPL {X  -159.990, Y  +469.047, Z    +0.000, E1   -66.225, E3 +146509.263}
SPL {X  -159.990, Y  +610.501, Z    +0.000, E1   -69.067, E3 +146596.867}
SPL {X  -159.990, Y  +630.690, Z    +0.000, E1   -69.080, E3 +146613.247}
SPL {X  -159.990, Y  +648.088, Z    +0.000, E1   -69.056, E3 +146627.423}
SPL {X  -159.990, Y  +663.340, Z    +0.000, E1   -69.061, E3 +146639.809}
SPL {X  -159.945, Y  +675.309, Z    +0.000, E1   -69.039, E3 +146649.621}
SPL {X  -159.172, Y  +687.655, Z    +0.000, E1   -68.973, E3 +146660.391}
SPL {X  -157.106, Y  +701.739, Z    +0.000, E1   -68.720, E3 +146674.000}
SPL {X  -154.598, Y  +712.687, Z    +0.000, E1   -68.393, E3 +146685.514}
SPL {X  -151.859, Y  +721.854, Z    +0.000, E1   -68.046, E3 +146695.734}
SPL {X  -148.628, Y  +730.715, Z    +0.000, E1   -67.614, E3 +146706.143}
SPL {X  -145.416, Y  +738.215, Z    +0.000, E1   -67.166, E3 +146715.351}
SPL {X  -142.090, Y  +745.034, Z    +0.000, E1   -66.692, E3 +146724.007}
SPL {X  -138.343, Y  +751.861, Z    +0.000, E1   -66.137, E3 +146732.934}
SPL {X  -134.819, Y  +757.643, Z    +0.000, E1   -65.575, E3 +146740.700}
SPL {X  -131.187, Y  +763.079, Z    +0.000, E1   -64.994, E3 +146748.083}
SPL {X  -127.405, Y  +768.272, Z    +0.000, E1   -64.349, E3 +146755.203}
SPL {X   -94.830, Y  +800.357, Z    +0.000, E1   -53.815, E3 +146869.736}
ENDSPLINE

SPLINE
SPL {X  -133.930, Y  +759.019, Z    +0.000, E1   -46.142, E3 +147017.119}
SPL {X  -149.331, Y  +728.920, Z    +0.000, E1   -37.154, E3 +147034.290}
SPL {X  -155.856, Y  +707.636, Z    +0.000, E1   -27.210, E3 +147040.293}
SPL {X  -159.260, Y  +686.764, Z    +0.000, E1   -14.026, E3 +147043.568}
SPL {X  -159.985, Y  +672.780, Z    +0.000, E1    -3.059, E3 +147044.469}
SPL {X  -159.990, Y  +669.259, Z    +0.000, E1    +0.225, E3 +147044.524}
SPL {X  -159.990, Y  +665.054, Z    +0.000, E1    +7.292, E3 +147044.629}
SPL {X  -159.990, Y  +658.864, Z    +0.000, E1   +19.708, E3 +147045.017}
SPL {X  -159.990, Y  +650.462, Z    +0.000, E1   +35.240, E3 +147046.029}
SPL {X  -159.990, Y  +636.155, Z    +0.000, E1   +51.890, E3 +147048.926}
SPL {X  -159.990, Y  +583.574, Z    +0.000, E1   +66.740, E3 +147068.722}
SPL {X  -159.990, Y  +451.342, Z    +0.000, E1   +68.591, E3 +147154.414}
ENDSPLINE

SPLINE
SPL {X  -159.990, Y  +495.016, Z    +0.000, E1   +61.398, E3 +147168.379}
ENDSPLINE

SPLINE
SPL {X  -159.990, Y  +469.556, Z    +0.000, E1   +62.943, E3 +147185.818}
SPL {X  -159.990, Y  +452.168, Z    +0.000, E1   +63.738, E3 +147198.374}
SPL {X  -159.990, Y  +433.781, Z    +0.000, E1   +64.535, E3 +147211.399}
SPL {X  -159.990, Y  +407.091, Z    +0.000, E1   +65.705, E3 +147228.602}
SPL {X  -159.990, Y  +383.383, Z    +0.000, E1   +66.590, E3 +147243.737}
SPL {X  -159.086, Y  +365.512, Z    +0.000, E1   +67.201, E3 +147254.834}
SPL {X  -155.924, Y  +346.662, Z    +0.000, E1   +68.026, E3 +147264.352}
SPL {X  -152.004, Y  +332.585, Z    +0.000, E1   +68.049, E3 +147275.790}
SPL {X  -147.728, Y  +321.072, Z    +0.000, E1   +67.490, E3 +147289.371}
SPL {X  -142.939, Y  +310.631, Z    +0.000, E1   +66.808, E3 +147302.438}
SPL {X  -138.502, Y  +302.413, Z    +0.000, E1   +66.138, E3 +147313.181}
SPL {X  -133.815, Y  +294.806, Z    +0.000, E1   +65.413, E3 +147323.387}
SPL {X  -130.038, Y  +289.296, Z    +0.000, E1   +64.749, E3 +147330.979}
SPL {X  -127.114, Y  +285.347, Z    +0.000, E1   +64.250, E3 +147336.402}
SPL {X   -96.237, Y  +254.690, Z    +0.000, E1   +52.223, E3 +147479.790}
ENDSPLINE

SPLINE
SPL {X  -139.640, Y  +304.414, Z    +0.000, E1   +43.367, E3 +147600.151}
SPL {X  -151.122, Y  +329.974, Z    +0.000, E1   +34.701, E3 +147612.942}
SPL {X  -155.699, Y  +345.695, Z    +0.000, E1   +27.167, E3 +147617.323}
SPL {X  -158.589, Y  +361.372, Z    +0.000, E1   +17.765, E3 +147620.088}
SPL {X  -159.702, Y  +372.901, Z    +0.000, E1    +9.563, E3 +147621.320}
SPL {X  -159.980, Y  +380.731, Z    +0.000, E1    +3.359, E3 +147621.717}
SPL {X  -159.990, Y  +384.465, Z    +0.000, E1    +0.049, E3 +147621.775}
SPL {X  -159.990, Y  +385.295, Z    +0.000, E1    -1.130, E3 +147621.780}
SPL {X  -159.990, Y  +387.941, Z    +0.000, E1    -5.453, E3 +147621.844}
SPL {X  -159.990, Y  +392.683, Z    +0.000, E1   -14.335, E3 +147622.102}
SPL {X  -159.990, Y  +399.462, Z    +0.000, E1   -27.551, E3 +147622.788}
SPL {X  -159.990, Y  +406.707, Z    +0.000, E1   -39.277, E3 +147623.943}
SPL {X  -159.990, Y  +418.467, Z    +0.000, E1   -51.591, E3 +147626.549}
SPL {X  -159.990, Y  +469.047, Z    +0.000, E1   -66.225, E3 +147645.626}
SPL {X  -159.990, Y  +610.501, Z    +0.000, E1   -69.067, E3 +147733.230}
SPL {X  -159.990, Y  +630.690, Z    +0.000, E1   -69.080, E3 +147749.611}
SPL {X  -159.990, Y  +652.219, Z    +0.000, E1   -69.078, E3 +147767.095}
SPL {X  -159.990, Y  +671.254, Z    +0.000, E1   -69.063, E3 +147782.596}
SPL {X  -159.471, Y  +684.377, Z    +0.000, E1   -68.989, E3 +147793.823}
SPL {X  -158.115, Y  +695.924, Z    +0.000, E1   -68.836, E3 +147804.607}
SPL {X  -156.463, Y  +704.909, Z    +0.000, E1   -68.615, E3 +147813.664}
SPL {X  -154.598, Y  +712.687, Z    +0.000, E1   -68.393, E3 +147821.878}
SPL {X  -151.859, Y  +721.854, Z    +0.000, E1   -68.046, E3 +147832.097}
SPL {X  -148.628, Y  +730.715, Z    +0.000, E1   -67.614, E3 +147842.506}
SPL {X  -145.416, Y  +738.215, Z    +0.000, E1   -67.166, E3 +147851.715}
SPL {X  -141.128, Y  +746.863, Z    +0.000, E1   -66.582, E3 +147862.692}
SPL {X  -137.485, Y  +753.321, Z    +0.000, E1   -65.984, E3 +147871.268}
SPL {X  -134.819, Y  +757.643, Z    +0.000, E1   -65.575, E3 +147877.063}
SPL {X  -131.187, Y  +763.079, Z    +0.000, E1   -64.994, E3 +147884.447}
SPL {X  -127.405, Y  +768.272, Z    +0.000, E1   -64.349, E3 +147891.567}
SPL {X   -94.830, Y  +800.357, Z    +0.000, E1   -53.815, E3 +148006.099}
ENDSPLINE

SPLINE
SPL {X  -133.930, Y  +759.019, Z    +0.000, E1   -46.142, E3 +148153.483}
SPL {X  -149.331, Y  +728.920, Z    +0.000, E1   -37.154, E3 +148170.653}
SPL {X  -155.856, Y  +707.636, Z    +0.000, E1   -27.210, E3 +148176.656}
SPL {X  -158.677, Y  +691.955, Z    +0.000, E1   -17.570, E3 +148179.362}
SPL {X  -159.802, Y  +679.261, Z    +0.000, E1    -8.330, E3 +148180.559}
SPL {X  -159.990, Y  +671.355, Z    +0.000, E1    -1.732, E3 +148180.869}
SPL {X  -159.990, Y  +669.500, Z    +0.000, E1    +0.000, E3 +148180.886}
SPL {X  -159.990, Y  +667.882, Z    +0.000, E1    +2.380, E3 +148180.905}
SPL {X  -159.990, Y  +664.041, Z    +0.000, E1    +9.423, E3 +148181.031}
SPL {X  -159.990, Y  +658.864, Z    +0.000, E1   +19.708, E3 +148181.381}
SPL {X  -159.990, Y  +650.462, Z    +0.000, E1   +35.240, E3 +148182.392}
SPL {X  -159.990, Y  +636.155, Z    +0.000, E1   +51.890, E3 +148185.290}
SPL {X  -159.990, Y  +583.574, Z    +0.000, E1   +66.740, E3 +148205.086}
SPL {X  -159.990, Y  +451.342, Z    +0.000, E1   +68.591, E3 +148290.778}
ENDSPLINE

SPLINE
SPL {X  -159.990, Y  +495.016, Z    +0.000, E1   +61.398, E3 +148304.742}
ENDSPLINE

SPLINE
SPL {X  -159.990, Y  +473.575, Z    +0.000, E1   +62.704, E3 +148319.477}
SPL {X  -159.990, Y  +455.620, Z    +0.000, E1   +63.615, E3 +148332.095}
SPL {X  -159.990, Y  +433.781, Z    +0.000, E1   +64.535, E3 +148347.762}
SPL {X  -159.990, Y  +407.091, Z    +0.000, E1   +65.705, E3 +148364.966}
SPL {X  -159.990, Y  +383.383, Z    +0.000, E1   +66.590, E3 +148380.100}
SPL {X  -158.268, Y  +359.089, Z    +0.000, E1   +67.514, E3 +148394.301}
SPL {X  -153.587, Y  +337.689, Z    +0.000, E1   +68.173, E3 +148407.035}
SPL {X  -150.185, Y  +327.353, Z    +0.000, E1   +67.790, E3 +148418.267}
SPL {X  -147.824, Y  +321.305, Z    +0.000, E1   +67.459, E3 +148425.531}
SPL {X  -144.736, Y  +314.321, Z    +0.000, E1   +67.058, E3 +148434.127}
SPL {X  -140.646, Y  +306.241, Z    +0.000, E1   +66.458, E3 +148444.506}
SPL {X  -136.388, Y  +298.863, Z    +0.000, E1   +65.814, E3 +148454.279}
SPL {X  -132.805, Y  +293.283, Z    +0.000, E1   +65.214, E3 +148461.868}
SPL {X  -130.038, Y  +289.296, Z    +0.000, E1   +64.749, E3 +148467.342}
SPL {X  -127.114, Y  +285.347, Z    +0.000, E1   +64.250, E3 +148472.765}
SPL {X   -96.237, Y  +254.690, Z    +0.000, E1   +52.223, E3 +148616.153}
ENDSPLINE

SPLINE
SPL {X  -139.640, Y  +304.414, Z    +0.000, E1   +43.367, E3 +148736.514}
SPL {X  -154.086, Y  +339.440, Z    +0.000, E1   +30.439, E3 +148752.072}
SPL {X  -158.589, Y  +361.372, Z    +0.000, E1   +17.765, E3 +148756.451}
SPL {X  -159.702, Y  +372.901, Z    +0.000, E1    +9.563, E3 +148757.683}
SPL {X  -159.980, Y  +380.731, Z    +0.000, E1    +3.359, E3 +148758.081}
SPL {X  -159.990, Y  +384.465, Z    +0.000, E1    +0.049, E3 +148758.138}
SPL {X  -159.990, Y  +386.161, Z    +0.000, E1    -2.359, E3 +148758.161}
SPL {X  -159.990, Y  +390.716, Z    +0.000, E1   -10.524, E3 +148758.336}
SPL {X  -159.990, Y  +397.792, Z    +0.000, E1   -24.215, E3 +148758.966}
SPL {X  -159.990, Y  +406.707, Z    +0.000, E1   -39.277, E3 +148760.307}
SPL {X  -159.990, Y  +418.467, Z    +0.000, E1   -51.591, E3 +148762.913}
SPL {X  -159.990, Y  +469.047, Z    +0.000, E1   -66.225, E3 +148781.990}
SPL {X  -159.990, Y  +610.501, Z    +0.000, E1   -69.067, E3 +148869.594}
SPL {X  -159.990, Y  +630.690, Z    +0.000, E1   -69.080, E3 +148885.974}
SPL {X  -159.990, Y  +652.219, Z    +0.000, E1   -69.078, E3 +148903.459}
SPL {X  -159.990, Y  +671.254, Z    +0.000, E1   -69.063, E3 +148918.959}
SPL {X  -159.172, Y  +687.655, Z    +0.000, E1   -68.973, E3 +148933.119}
SPL {X  -157.106, Y  +701.739, Z    +0.000, E1   -68.720, E3 +148946.727}
SPL {X  -154.598, Y  +712.687, Z    +0.000, E1   -68.393, E3 +148958.242}
SPL {X  -151.859, Y  +721.854, Z    +0.000, E1   -68.046, E3 +148968.461}
SPL {X  -148.628, Y  +730.715, Z    +0.000, E1   -67.614, E3 +148978.870}
SPL {X  -145.416, Y  +738.215, Z    +0.000, E1   -67.166, E3 +148988.078}
SPL {X  -141.128, Y  +746.863, Z    +0.000, E1   -66.582, E3 +148999.055}
SPL {X  -137.485, Y  +753.321, Z    +0.000, E1   -65.984, E3 +149007.632}
SPL {X  -134.819, Y  +757.643, Z    +0.000, E1   -65.575, E3 +149013.427}
SPL {X  -131.187, Y  +763.079, Z    +0.000, E1   -64.994, E3 +149020.810}
SPL {X  -127.405, Y  +768.272, Z    +0.000, E1   -64.349, E3 +149027.931}
SPL {X   -94.830, Y  +800.357, Z    +0.000, E1   -53.815, E3 +149142.463}
ENDSPLINE

SPLINE
SPL {X  -133.930, Y  +759.019, Z    +0.000, E1   -46.142, E3 +149289.846}
SPL {X  -149.331, Y  +728.920, Z    +0.000, E1   -37.154, E3 +149307.017}
SPL {X  -155.856, Y  +707.636, Z    +0.000, E1   -27.210, E3 +149313.020}
SPL {X  -158.677, Y  +691.955, Z    +0.000, E1   -17.570, E3 +149315.726}
SPL {X  -159.802, Y  +679.261, Z    +0.000, E1    -8.330, E3 +149316.922}
SPL {X  -159.990, Y  +671.355, Z    +0.000, E1    -1.732, E3 +149317.232}
SPL {X  -159.990, Y  +669.500, Z    +0.000, E1    +0.000, E3 +149317.250}
SPL {X  -159.990, Y  +667.882, Z    +0.000, E1    +2.380, E3 +149317.269}
SPL {X  -159.990, Y  +664.041, Z    +0.000, E1    +9.423, E3 +149317.395}
SPL {X  -159.990, Y  +658.864, Z    +0.000, E1   +19.708, E3 +149317.745}
SPL {X  -159.990, Y  +650.462, Z    +0.000, E1   +35.240, E3 +149318.756}
SPL {X  -159.990, Y  +636.155, Z    +0.000, E1   +51.890, E3 +149321.653}
SPL {X  -159.990, Y  +583.574, Z    +0.000, E1   +66.740, E3 +149341.450}
SPL {X  -159.990, Y  +451.342, Z    +0.000, E1   +68.591, E3 +149427.141}
ENDSPLINE

SPLINE
SPL {X  -159.990, Y  +495.016, Z    +0.000, E1   +61.398, E3 +149441.106}
ENDSPLINE

SPLINE
SPL {X  -159.990, Y  +473.575, Z    +0.000, E1   +62.704, E3 +149455.841}
SPL {X  -159.990, Y  +455.620, Z    +0.000, E1   +63.615, E3 +149468.459}
SPL {X  -159.990, Y  +433.781, Z    +0.000, E1   +64.535, E3 +149484.126}
SPL {X  -159.990, Y  +407.091, Z    +0.000, E1   +65.705, E3 +149501.330}
SPL {X  -159.990, Y  +383.383, Z    +0.000, E1   +66.590, E3 +149516.464}
SPL {X  -158.268, Y  +359.089, Z    +0.000, E1   +67.514, E3 +149530.665}
SPL {X  -153.587, Y  +337.689, Z    +0.000, E1   +68.173, E3 +149543.399}
SPL {X  -150.185, Y  +327.353, Z    +0.000, E1   +67.790, E3 +149554.631}
SPL {X  -147.050, Y  +319.468, Z    +0.000, E1   +67.370, E3 +149564.112}
SPL {X  -142.939, Y  +310.631, Z    +0.000, E1   +66.808, E3 +149575.166}
SPL {X  -138.502, Y  +302.413, Z    +0.000, E1   +66.138, E3 +149585.908}
SPL {X  -135.296, Y  +297.108, Z    +0.000, E1   +65.610, E3 +149593.048}
SPL {X  -132.805, Y  +293.283, Z    +0.000, E1   +65.214, E3 +149598.232}
SPL {X  -130.038, Y  +289.296, Z    +0.000, E1   +64.749, E3 +149603.706}
SPL {X  -127.114, Y  +285.347, Z    +0.000, E1   +64.250, E3 +149609.129}
SPL {X   -96.237, Y  +254.690, Z    +0.000, E1   +52.223, E3 +149752.517}
ENDSPLINE

SPLINE
SPL {X  -139.640, Y  +304.414, Z    +0.000, E1   +43.367, E3 +149872.878}
SPL {X  -154.086, Y  +339.440, Z    +0.000, E1   +30.439, E3 +149888.435}
SPL {X  -158.589, Y  +361.372, Z    +0.000, E1   +17.765, E3 +149892.815}
SPL {X  -159.702, Y  +372.901, Z    +0.000, E1    +9.563, E3 +149894.047}
SPL {X  -159.980, Y  +380.731, Z    +0.000, E1    +3.359, E3 +149894.445}
SPL {X  -159.990, Y  +384.465, Z    +0.000, E1    +0.049, E3 +149894.502}
SPL {X  -159.990, Y  +386.161, Z    +0.000, E1    -2.359, E3 +149894.525}
SPL {X  -159.990, Y  +391.786, Z    +0.000, E1   -12.382, E3 +149894.775}
SPL {X  -159.990, Y  +399.462, Z    +0.000, E1   -27.551, E3 +149895.515}
SPL {X  -159.990, Y  +406.707, Z    +0.000, E1   -39.277, E3 +149896.671}
SPL {X  -159.990, Y  +418.467, Z    +0.000, E1   -51.591, E3 +149899.276}
SPL {X  -159.990, Y  +469.047, Z    +0.000, E1   -66.225, E3 +149918.354}
SPL {X  -159.990, Y  +610.501, Z    +0.000, E1   -69.067, E3 +150005.957}
SPL {X  -159.990, Y  +623.913, Z    +0.000, E1   -69.046, E3 +150016.906}
SPL {X  -159.990, Y  +635.131, Z    +0.000, E1   -69.053, E3 +150026.007}
SPL {X  -159.990, Y  +648.088, Z    +0.000, E1   -69.056, E3 +150036.514}
SPL {X  -159.990, Y  +667.800, Z    +0.000, E1   -69.089, E3 +150052.463}
SPL {X  -159.172, Y  +687.655, Z    +0.000, E1   -68.973, E3 +150069.482}
SPL {X  -157.106, Y  +701.739, Z    +0.000, E1   -68.720, E3 +150083.091}
SPL {X  -154.598, Y  +712.687, Z    +0.000, E1   -68.393, E3 +150094.605}
SPL {X  -151.859, Y  +721.854, Z    +0.000, E1   -68.046, E3 +150104.824}
SPL {X  -148.628, Y  +730.715, Z    +0.000, E1   -67.614, E3 +150115.234}
SPL {X  -145.416, Y  +738.215, Z    +0.000, E1   -67.166, E3 +150124.442}
SPL {X  -142.090, Y  +745.034, Z    +0.000, E1   -66.692, E3 +150133.098}
SPL {X  -138.343, Y  +751.861, Z    +0.000, E1   -66.137, E3 +150142.025}
SPL {X  -134.819, Y  +757.643, Z    +0.000, E1   -65.575, E3 +150149.791}
SPL {X  -131.187, Y  +763.079, Z    +0.000, E1   -64.994, E3 +150157.174}
SPL {X  -127.405, Y  +768.272, Z    +0.000, E1   -64.349, E3 +150164.294}
SPL {X   -94.830, Y  +800.357, Z    +0.000, E1   -53.815, E3 +150278.827}
ENDSPLINE

SPLINE
SPL {X  -133.930, Y  +759.019, Z    +0.000, E1   -46.142, E3 +150426.210}
SPL {X  -149.331, Y  +728.920, Z    +0.000, E1   -37.154, E3 +150443.381}
SPL {X  -155.856, Y  +707.636, Z    +0.000, E1   -27.210, E3 +150449.384}
SPL {X  -158.677, Y  +691.955, Z    +0.000, E1   -17.570, E3 +150452.090}
SPL {X  -159.802, Y  +679.261, Z    +0.000, E1    -8.330, E3 +150453.286}
SPL {X  -159.990, Y  +669.767, Z    +0.000, E1    -0.394, E3 +150453.611}
SPL {X  -159.990, Y  +667.882, Z    +0.000, E1    +2.380, E3 +150453.633}
SPL {X  -159.990, Y  +664.041, Z    +0.000, E1    +9.423, E3 +150453.759}
SPL {X  -159.990, Y  +658.864, Z    +0.000, E1   +19.708, E3 +150454.108}
SPL {X  -159.990, Y  +650.462, Z    +0.000, E1   +35.240, E3 +150455.120}
SPL {X  -159.990, Y  +636.155, Z    +0.000, E1   +51.890, E3 +150458.017}
SPL {X  -159.990, Y  +583.574, Z    +0.000, E1   +66.740, E3 +150477.813}
SPL {X  -159.990, Y  +451.342, Z    +0.000, E1   +68.591, E3 +150563.505}
ENDSPLINE

SPLINE
SPL {X  -159.990, Y  +495.016, Z    +0.000, E1   +61.398, E3 +150577.470}
ENDSPLINE

SPLINE
SPL {X  -159.990, Y  +469.556, Z    +0.000, E1   +62.943, E3 +150594.909}
SPL {X  -159.990, Y  +452.168, Z    +0.000, E1   +63.738, E3 +150607.464}
SPL {X  -159.990, Y  +433.781, Z    +0.000, E1   +64.535, E3 +150620.490}
SPL {X  -159.990, Y  +407.091, Z    +0.000, E1   +65.705, E3 +150637.693}
SPL {X  -159.990, Y  +383.383, Z    +0.000, E1   +66.590, E3 +150652.828}
SPL {X  -159.086, Y  +365.512, Z    +0.000, E1   +67.201, E3 +150663.925}
SPL {X  -155.924, Y  +346.662, Z    +0.000, E1   +68.026, E3 +150673.442}
SPL {X  -152.004, Y  +332.585, Z    +0.000, E1   +68.049, E3 +150684.881}
SPL {X  -147.728, Y  +321.072, Z    +0.000, E1   +67.490, E3 +150698.462}
SPL {X  -142.939, Y  +310.631, Z    +0.000, E1   +66.808, E3 +150711.529}
SPL {X  -138.502, Y  +302.413, Z    +0.000, E1   +66.138, E3 +150722.272}
SPL {X  -135.296, Y  +297.108, Z    +0.000, E1   +65.610, E3 +150729.412}
SPL {X  -132.805, Y  +293.283, Z    +0.000, E1   +65.214, E3 +150734.595}
SPL {X  -130.038, Y  +289.296, Z    +0.000, E1   +64.749, E3 +150740.070}
SPL {X  -127.114, Y  +285.347, Z    +0.000, E1   +64.250, E3 +150745.493}
SPL {X   -96.237, Y  +254.690, Z    +0.000, E1   +52.223, E3 +150888.881}
ENDSPLINE

SPLINE
SPL {X  -139.640, Y  +304.414, Z    +0.000, E1   +43.367, E3 +151009.242}
SPL {X  -151.122, Y  +329.974, Z    +0.000, E1   +34.701, E3 +151022.033}
SPL {X  -155.699, Y  +345.695, Z    +0.000, E1   +27.167, E3 +151026.414}
SPL {X  -158.589, Y  +361.372, Z    +0.000, E1   +17.765, E3 +151029.179}
SPL {X  -159.702, Y  +372.901, Z    +0.000, E1    +9.563, E3 +151030.411}
SPL {X  -159.980, Y  +380.731, Z    +0.000, E1    +3.359, E3 +151030.808}
SPL {X  -159.990, Y  +384.465, Z    +0.000, E1    +0.049, E3 +151030.866}
SPL {X  -159.990, Y  +386.161, Z    +0.000, E1    -2.359, E3 +151030.888}
SPL {X  -159.990, Y  +391.786, Z    +0.000, E1   -12.382, E3 +151031.139}
SPL {X  -159.990, Y  +399.462, Z    +0.000, E1   -27.551, E3 +151031.879}
SPL {X  -159.990, Y  +406.707, Z    +0.000, E1   -39.277, E3 +151033.034}
SPL {X  -159.990, Y  +418.467, Z    +0.000, E1   -51.591, E3 +151035.640}
SPL {X  -159.990, Y  +469.047, Z    +0.000, E1   -66.225, E3 +151054.717}
SPL {X  -159.990, Y  +610.501, Z    +0.000, E1   -69.067, E3 +151142.321}
SPL {X  -159.990, Y  +623.913, Z    +0.000, E1   -69.046, E3 +151153.270}
SPL {X  -159.990, Y  +635.131, Z    +0.000, E1   -69.053, E3 +151162.371}
SPL {X  -159.990, Y  +648.088, Z    +0.000, E1   -69.056, E3 +151172.878}
SPL {X  -159.990, Y  +663.340, Z    +0.000, E1   -69.061, E3 +151185.264}
SPL {X  -159.706, Y  +681.022, Z    +0.000, E1   -69.040, E3 +151199.896}
SPL {X  -158.115, Y  +695.924, Z    +0.000, E1   -68.836, E3 +151213.697}
SPL {X  -156.463, Y  +704.909, Z    +0.000, E1   -68.615, E3 +151222.755}
SPL {X  -154.598, Y  +712.687, Z    +0.000, E1   -68.393, E3 +151230.969}
SPL {X  -151.859, Y  +721.854, Z    +0.000, E1   -68.046, E3 +151241.188}
SPL {X  -148.628, Y  +730.715, Z    +0.000, E1   -67.614, E3 +151251.597}
SPL {X  -145.416, Y  +738.215, Z    +0.000, E1   -67.166, E3 +151260.806}
SPL {X  -142.090, Y  +745.034, Z    +0.000, E1   -66.692, E3 +151269.461}
SPL {X  -138.343, Y  +751.861, Z    +0.000, E1   -66.137, E3 +151278.388}
SPL {X  -134.819, Y  +757.643, Z    +0.000, E1   -65.575, E3 +151286.154}
SPL {X  -131.187, Y  +763.079, Z    +0.000, E1   -64.994, E3 +151293.538}
SPL {X  -127.405, Y  +768.272, Z    +0.000, E1   -64.349, E3 +151300.658}
SPL {X   -94.830, Y  +800.357, Z    +0.000, E1   -53.815, E3 +151415.190}
ENDSPLINE

SPLINE
SPL {X  -133.930, Y  +759.019, Z    +0.000, E1   -46.142, E3 +151562.574}
SPL {X  -149.331, Y  +728.920, Z    +0.000, E1   -37.154, E3 +151579.744}
SPL {X  -155.856, Y  +707.636, Z    +0.000, E1   -27.210, E3 +151585.747}
SPL {X  -158.677, Y  +691.955, Z    +0.000, E1   -17.570, E3 +151588.453}
SPL {X  -159.802, Y  +679.261, Z    +0.000, E1    -8.330, E3 +151589.650}
SPL {X  -159.990, Y  +669.767, Z    +0.000, E1    -0.394, E3 +151589.974}
SPL {X  -159.990, Y  +667.882, Z    +0.000, E1    +2.380, E3 +151589.996}
SPL {X  -159.990, Y  +664.041, Z    +0.000, E1    +9.423, E3 +151590.122}
SPL {X  -159.990, Y  +660.147, Z    +0.000, E1   +17.275, E3 +151590.360}
SPL {X  -159.990, Y  +656.649, Z    +0.000, E1   +24.355, E3 +151590.666}
SPL {X  -159.990, Y  +650.462, Z    +0.000, E1   +35.240, E3 +151591.483}
SPL {X  -159.990, Y  +636.155, Z    +0.000, E1   +51.890, E3 +151594.381}
SPL {X  -159.990, Y  +583.574, Z    +0.000, E1   +66.740, E3 +151614.177}
SPL {X  -159.990, Y  +451.342, Z    +0.000, E1   +68.591, E3 +151699.869}
ENDSPLINE

SPLINE
SPL {X  -159.990, Y  +495.016, Z    +0.000, E1   +61.398, E3 +151713.833}
ENDSPLINE

SPLINE
SPL {X  -159.990, Y  +473.575, Z    +0.000, E1   +62.704, E3 +151728.568}
SPL {X  -159.990, Y  +455.620, Z    +0.000, E1   +63.615, E3 +151741.186}
SPL {X  -159.990, Y  +439.579, Z    +0.000, E1   +64.263, E3 +151752.921}
SPL {X  -159.990, Y  +420.812, Z    +0.000, E1   +65.111, E3 +151765.353}
SPL {X  -159.990, Y  +400.802, Z    +0.000, E1   +65.940, E3 +151778.094}
SPL {X  -159.990, Y  +383.383, Z    +0.000, E1   +66.590, E3 +151789.191}
SPL {X  -159.086, Y  +365.512, Z    +0.000, E1   +67.201, E3 +151800.289}
SPL {X  -155.924, Y  +346.662, Z    +0.000, E1   +68.026, E3 +151809.806}
SPL {X  -152.751, Y  +334.918, Z    +0.000, E1   +68.124, E3 +151818.636}
SPL {X  -150.185, Y  +327.353, Z    +0.000, E1   +67.790, E3 +151827.358}
SPL {X  -147.050, Y  +319.468, Z    +0.000, E1   +67.370, E3 +151836.839}
SPL {X  -143.990, Y  +312.760, Z    +0.000, E1   +66.929, E3 +151845.228}
SPL {X  -140.646, Y  +306.241, Z    +0.000, E1   +66.458, E3 +151853.597}
SPL {X  -137.570, Y  +300.823, Z    +0.000, E1   +65.968, E3 +151860.788}
SPL {X  -133.815, Y  +294.806, Z    +0.000, E1   +65.413, E3 +151868.842}
SPL {X  -130.038, Y  +289.296, Z    +0.000, E1   +64.749, E3 +151876.433}
SPL {X  -127.114, Y  +285.347, Z    +0.000, E1   +64.250, E3 +151881.856}
SPL {X   -96.237, Y  +254.690, Z    +0.000, E1   +52.223, E3 +152025.244}
ENDSPLINE

SPLINE
SPL {X  -139.640, Y  +304.414, Z    +0.000, E1   +43.367, E3 +152145.605}
SPL {X  -151.122, Y  +329.974, Z    +0.000, E1   +34.701, E3 +152158.397}
SPL {X  -155.699, Y  +345.695, Z    +0.000, E1   +27.167, E3 +152162.778}
SPL {X  -158.589, Y  +361.372, Z    +0.000, E1   +17.765, E3 +152165.542}
SPL {X  -159.702, Y  +372.901, Z    +0.000, E1    +9.563, E3 +152166.774}
SPL {X  -159.980, Y  +380.731, Z    +0.000, E1    +3.359, E3 +152167.172}
SPL {X  -159.990, Y  +384.465, Z    +0.000, E1    +0.049, E3 +152167.229}
SPL {X  -159.990, Y  +386.161, Z    +0.000, E1    -2.359, E3 +152167.252}
SPL {X  -159.990, Y  +391.786, Z    +0.000, E1   -12.382, E3 +152167.503}
SPL {X  -159.990, Y  +399.462, Z    +0.000, E1   -27.551, E3 +152168.242}
SPL {X  -159.990, Y  +406.707, Z    +0.000, E1   -39.277, E3 +152169.398}
SPL {X  -159.990, Y  +418.467, Z    +0.000, E1   -51.591, E3 +152172.004}
SPL {X  -159.990, Y  +469.047, Z    +0.000, E1   -66.225, E3 +152191.081}
SPL {X  -159.990, Y  +610.501, Z    +0.000, E1   -69.067, E3 +152278.685}
SPL {X  -159.990, Y  +623.913, Z    +0.000, E1   -69.046, E3 +152289.633}
SPL {X  -159.990, Y  +635.131, Z    +0.000, E1   -69.053, E3 +152298.734}
SPL {X  -159.990, Y  +648.088, Z    +0.000, E1   -69.056, E3 +152309.241}
SPL {X  -159.990, Y  +663.340, Z    +0.000, E1   -69.061, E3 +152321.627}
SPL {X  -159.706, Y  +681.022, Z    +0.000, E1   -69.040, E3 +152336.260}
SPL {X  -158.115, Y  +695.924, Z    +0.000, E1   -68.836, E3 +152350.061}
SPL {X  -156.463, Y  +704.909, Z    +0.000, E1   -68.615, E3 +152359.119}
SPL {X  -154.598, Y  +712.687, Z    +0.000, E1   -68.393, E3 +152367.333}
SPL {X  -151.859, Y  +721.854, Z    +0.000, E1   -68.046, E3 +152377.552}
SPL {X  -148.628, Y  +730.715, Z    +0.000, E1   -67.614, E3 +152387.961}
SPL {X  -145.416, Y  +738.215, Z    +0.000, E1   -67.166, E3 +152397.169}
SPL {X  -142.090, Y  +745.034, Z    +0.000, E1   -66.692, E3 +152405.825}
SPL {X  -138.343, Y  +751.861, Z    +0.000, E1   -66.137, E3 +152414.752}
SPL {X  -134.819, Y  +757.643, Z    +0.000, E1   -65.575, E3 +152422.518}
SPL {X  -131.187, Y  +763.079, Z    +0.000, E1   -64.994, E3 +152429.901}
SPL {X  -127.405, Y  +768.272, Z    +0.000, E1   -64.349, E3 +152437.022}
SPL {X   -94.830, Y  +800.357, Z    +0.000, E1   -53.815, E3 +152551.554}
ENDSPLINE

SPLINE
SPL {X  -133.930, Y  +759.019, Z    +0.000, E1   -46.142, E3 +152698.937}
SPL {X  -149.331, Y  +728.920, Z    +0.000, E1   -37.154, E3 +152716.108}
SPL {X  -155.856, Y  +707.636, Z    +0.000, E1   -27.210, E3 +152722.111}
SPL {X  -159.260, Y  +686.764, Z    +0.000, E1   -14.026, E3 +152725.386}
SPL {X  -159.985, Y  +672.780, Z    +0.000, E1    -3.059, E3 +152726.287}
SPL {X  -159.990, Y  +669.259, Z    +0.000, E1    +0.225, E3 +152726.342}
SPL {X  -159.990, Y  +665.054, Z    +0.000, E1    +7.292, E3 +152726.447}
SPL {X  -159.990, Y  +658.864, Z    +0.000, E1   +19.708, E3 +152726.836}
SPL {X  -159.990, Y  +650.462, Z    +0.000, E1   +35.240, E3 +152727.847}
SPL {X  -159.990, Y  +636.155, Z    +0.000, E1   +51.890, E3 +152730.744}
SPL {X  -159.990, Y  +583.574, Z    +0.000, E1   +66.740, E3 +152750.541}
SPL {X  -159.990, Y  +451.342, Z    +0.000, E1   +68.591, E3 +152836.232}
ENDSPLINE

SPLINE
SPL {X  -159.990, Y  +495.016, Z    +0.000, E1   +61.398, E3 +152850.197}
ENDSPLINE

SPLINE
SPL {X  -159.990, Y  +469.556, Z    +0.000, E1   +62.943, E3 +152867.636}
SPL {X  -159.990, Y  +452.168, Z    +0.000, E1   +63.738, E3 +152880.192}
SPL {X  -159.990, Y  +433.781, Z    +0.000, E1   +64.535, E3 +152893.217}
SPL {X  -159.990, Y  +414.623, Z    +0.000, E1   +65.374, E3 +152905.637}
SPL {X  -159.990, Y  +395.826, Z    +0.000, E1   +66.138, E3 +152917.652}
SPL {X  -159.536, Y  +370.459, Z    +0.000, E1   +67.052, E3 +152933.544}
SPL {X  -157.113, Y  +352.293, Z    +0.000, E1   +67.811, E3 +152943.126}
SPL {X  -153.587, Y  +337.689, Z    +0.000, E1   +68.173, E3 +152952.490}
SPL {X  -150.185, Y  +327.353, Z    +0.000, E1   +67.790, E3 +152963.722}
SPL {X  -147.824, Y  +321.305, Z    +0.000, E1   +67.459, E3 +152970.985}
SPL {X  -144.736, Y  +314.321, Z    +0.000, E1   +67.058, E3 +152979.582}
SPL {X  -141.667, Y  +308.155, Z    +0.000, E1   +66.586, E3 +152987.503}
SPL {X  -138.502, Y  +302.413, Z    +0.000, E1   +66.138, E3 +152994.999}
SPL {X  -135.296, Y  +297.108, Z    +0.000, E1   +65.610, E3 +153002.139}
SPL {X  -132.805, Y  +293.283, Z    +0.000, E1   +65.214, E3 +153007.323}
SPL {X  -130.038, Y  +289.296, Z    +0.000, E1   +64.749, E3 +153012.797}
SPL {X  -127.114, Y  +285.347, Z    +0.000, E1   +64.250, E3 +153018.220}
SPL {X   -96.237, Y  +254.690, Z    +0.000, E1   +52.223, E3 +153161.608}
ENDSPLINE

SPLINE
SPL {X  -139.640, Y  +304.414, Z    +0.000, E1   +43.367, E3 +153281.969}
SPL {X  -154.086, Y  +339.440, Z    +0.000, E1   +30.439, E3 +153297.526}
SPL {X  -158.589, Y  +361.372, Z    +0.000, E1   +17.765, E3 +153301.906}
SPL {X  -159.702, Y  +372.901, Z    +0.000, E1    +9.563, E3 +153303.138}
SPL {X  -159.980, Y  +380.731, Z    +0.000, E1    +3.359, E3 +153303.536}
SPL {X  -159.990, Y  +384.465, Z    +0.000, E1    +0.049, E3 +153303.593}
SPL {X  -159.990, Y  +385.295, Z    +0.000, E1    -1.130, E3 +153303.599}
SPL {X  -159.990, Y  +387.941, Z    +0.000, E1    -5.453, E3 +153303.662}
SPL {X  -159.990, Y  +392.683, Z    +0.000, E1   -14.335, E3 +153303.920}
SPL {X  -159.990, Y  +399.462, Z    +0.000, E1   -27.551, E3 +153304.606}
SPL {X  -159.990, Y  +406.707, Z    +0.000, E1   -39.277, E3 +153305.762}
SPL {X  -159.990, Y  +418.467, Z    +0.000, E1   -51.591, E3 +153308.367}
SPL {X  -159.990, Y  +469.047, Z    +0.000, E1   -66.225, E3 +153327.444}
SPL {X  -159.990, Y  +610.501, Z    +0.000, E1   -69.067, E3 +153415.048}
SPL {X  -159.990, Y  +623.913, Z    +0.000, E1   -69.046, E3 +153425.997}
SPL {X  -159.990, Y  +635.131, Z    +0.000, E1   -69.053, E3 +153435.098}
SPL {X  -159.990, Y  +648.088, Z    +0.000, E1   -69.056, E3 +153445.605}
SPL {X  -159.990, Y  +667.800, Z    +0.000, E1   -69.089, E3 +153461.554}
SPL {X  -159.471, Y  +684.377, Z    +0.000, E1   -68.989, E3 +153475.641}
SPL {X  -158.115, Y  +695.924, Z    +0.000, E1   -68.836, E3 +153486.425}
SPL {X  -156.463, Y  +704.909, Z    +0.000, E1   -68.615, E3 +153495.482}
SPL {X  -153.837, Y  +715.444, Z    +0.000, E1   -68.325, E3 +153506.660}
SPL {X  -151.088, Y  +724.124, Z    +0.000, E1   -67.925, E3 +153516.570}
SPL {X  -148.628, Y  +730.715, Z    +0.000, E1   -67.614, E3 +153524.325}
SPL {X  -145.416, Y  +738.215, Z    +0.000, E1   -67.166, E3 +153533.533}
SPL {X  -142.090, Y  +745.034, Z    +0.000, E1   -66.692, E3 +153542.189}
SPL {X  -138.343, Y  +751.861, Z    +0.000, E1   -66.137, E3 +153551.115}
SPL {X  -133.893, Y  +759.076, Z    +0.000, E1   -65.453, E3 +153560.791}
SPL {X  -130.341, Y  +764.280, Z    +0.000, E1   -64.831, E3 +153567.930}
SPL {X  -127.405, Y  +768.272, Z    +0.000, E1   -64.349, E3 +153573.385}
SPL {X   -94.830, Y  +800.357, Z    +0.000, E1   -53.815, E3 +153687.917}
ENDSPLINE

SPLINE
SPL {X  -133.930, Y  +759.019, Z    +0.000, E1   -46.142, E3 +153835.301}
SPL {X  -149.331, Y  +728.920, Z    +0.000, E1   -37.154, E3 +153852.471}
SPL {X  -155.856, Y  +707.636, Z    +0.000, E1   -27.210, E3 +153858.475}
SPL {X  -158.677, Y  +691.955, Z    +0.000, E1   -17.570, E3 +153861.180}
SPL {X  -159.802, Y  +679.261, Z    +0.000, E1    -8.330, E3 +153862.377}
SPL {X  -159.990, Y  +669.767, Z    +0.000, E1    -0.394, E3 +153862.702}
SPL {X  -159.990, Y  +667.882, Z    +0.000, E1    +2.380, E3 +153862.724}
SPL {X  -159.990, Y  +664.041, Z    +0.000, E1    +9.423, E3 +153862.850}
SPL {X  -159.990, Y  +660.147, Z    +0.000, E1   +17.275, E3 +153863.087}
SPL {X  -159.990, Y  +656.649, Z    +0.000, E1   +24.355, E3 +153863.393}
SPL {X  -159.990, Y  +650.462, Z    +0.000, E1   +35.240, E3 +153864.211}
SPL {X  -159.990, Y  +636.155, Z    +0.000, E1   +51.890, E3 +153867.108}
SPL {X  -159.990, Y  +583.574, Z    +0.000, E1   +66.740, E3 +153886.904}
SPL {X  -159.990, Y  +451.342, Z    +0.000, E1   +68.591, E3 +153972.596}
ENDSPLINE

SPLINE
SPL {X  -159.990, Y  +495.016, Z    +0.000, E1   +61.398, E3 +153986.561}
ENDSPLINE

SPLINE
SPL {X  -159.990, Y  +469.556, Z    +0.000, E1   +62.943, E3 +154004.000}
SPL {X  -159.990, Y  +445.297, Z    +0.000, E1   +64.051, E3 +154021.489}
SPL {X  -159.990, Y  +420.812, Z    +0.000, E1   +65.111, E3 +154038.080}
SPL {X  -159.990, Y  +395.826, Z    +0.000, E1   +66.138, E3 +154054.015}
SPL {X  -159.536, Y  +370.459, Z    +0.000, E1   +67.052, E3 +154069.908}
SPL {X  -155.924, Y  +346.662, Z    +0.000, E1   +68.026, E3 +154082.533}
SPL {X  -152.004, Y  +332.585, Z    +0.000, E1   +68.049, E3 +154093.971}
SPL {X  -148.519, Y  +323.011, Z    +0.000, E1   +67.572, E3 +154105.248}
SPL {X  -144.736, Y  +314.321, Z    +0.000, E1   +67.058, E3 +154115.945}
SPL {X  -140.646, Y  +306.241, Z    +0.000, E1   +66.458, E3 +154126.324}
SPL {X  -136.388, Y  +298.863, Z    +0.000, E1   +65.814, E3 +154136.097}
SPL {X  -132.805, Y  +293.283, Z    +0.000, E1   +65.214, E3 +154143.686}
SPL {X  -130.038, Y  +289.296, Z    +0.000, E1   +64.749, E3 +154149.160}
SPL {X  -127.114, Y  +285.347, Z    +0.000, E1   +64.250, E3 +154154.583}
SPL {X   -96.237, Y  +254.690, Z    +0.000, E1   +52.223, E3 +154297.972}
ENDSPLINE

SPLINE
SPL {X  -139.640, Y  +304.414, Z    +0.000, E1   +43.367, E3 +154418.332}
SPL {X  -154.086, Y  +339.440, Z    +0.000, E1   +30.439, E3 +154433.890}
SPL {X  -158.589, Y  +361.372, Z    +0.000, E1   +17.765, E3 +154438.270}
SPL {X  -159.702, Y  +372.901, Z    +0.000, E1    +9.563, E3 +154439.501}
SPL {X  -159.980, Y  +380.731, Z    +0.000, E1    +3.359, E3 +154439.899}
SPL {X  -159.990, Y  +384.708, Z    +0.000, E1    -0.166, E3 +154439.958}
SPL {X  -159.990, Y  +387.941, Z    +0.000, E1    -5.453, E3 +154440.026}
SPL {X  -159.990, Y  +391.582, Z    +0.000, E1   -12.331, E3 +154440.200}
SPL {X  -159.990, Y  +397.792, Z    +0.000, E1   -24.215, E3 +154440.784}
SPL {X  -159.990, Y  +406.707, Z    +0.000, E1   -39.277, E3 +154442.125}
SPL {X  -159.990, Y  +418.467, Z    +0.000, E1   -51.591, E3 +154444.731}
SPL {X  -159.990, Y  +469.047, Z    +0.000, E1   -66.225, E3 +154463.808}
SPL {X  -159.990, Y  +610.501, Z    +0.000, E1   -69.067, E3 +154551.412}
SPL {X  -159.990, Y  +623.913, Z    +0.000, E1   -69.046, E3 +154562.361}
SPL {X  -159.990, Y  +635.131, Z    +0.000, E1   -69.053, E3 +154571.462}
SPL {X  -159.990, Y  +652.219, Z    +0.000, E1   -69.078, E3 +154585.277}
SPL {X  -159.990, Y  +671.254, Z    +0.000, E1   -69.063, E3 +154600.778}
SPL {X  -159.471, Y  +684.377, Z    +0.000, E1   -68.989, E3 +154612.005}
SPL {X  -158.115, Y  +695.924, Z    +0.000, E1   -68.836, E3 +154622.788}
SPL {X  -156.463, Y  +704.909, Z    +0.000, E1   -68.615, E3 +154631.846}
SPL {X  -154.598, Y  +712.687, Z    +0.000, E1   -68.393, E3 +154640.060}
SPL {X  -151.859, Y  +721.854, Z    +0.000, E1   -68.046, E3 +154650.279}
SPL {X  -148.628, Y  +730.715, Z    +0.000, E1   -67.614, E3 +154660.688}
SPL {X  -145.416, Y  +738.215, Z    +0.000, E1   -67.166, E3 +154669.897}
SPL {X  -141.128, Y  +746.863, Z    +0.000, E1   -66.582, E3 +154680.874}
SPL {X  -137.485, Y  +753.321, Z    +0.000, E1   -65.984, E3 +154689.450}
SPL {X  -133.893, Y  +759.076, Z    +0.000, E1   -65.453, E3 +154697.155}
SPL {X  -130.341, Y  +764.280, Z    +0.000, E1   -64.831, E3 +154704.293}
SPL {X  -127.405, Y  +768.272, Z    +0.000, E1   -64.349, E3 +154709.749}
SPL {X   -94.830, Y  +800.357, Z    +0.000, E1   -53.815, E3 +154824.281}
ENDSPLINE

SPLINE
SPL {X  -133.930, Y  +759.019, Z    +0.000, E1   -46.142, E3 +154971.665}
SPL {X  -149.331, Y  +728.920, Z    +0.000, E1   -37.154, E3 +154988.835}
SPL {X  -155.856, Y  +707.636, Z    +0.000, E1   -27.210, E3 +154994.838}
SPL {X  -158.677, Y  +691.955, Z    +0.000, E1   -17.570, E3 +154997.544}
SPL {X  -159.802, Y  +679.261, Z    +0.000, E1    -8.330, E3 +154998.741}
SPL {X  -159.990, Y  +669.767, Z    +0.000, E1    -0.394, E3 +154999.065}
SPL {X  -159.990, Y  +667.882, Z    +0.000, E1    +2.380, E3 +154999.087}
SPL {X  -159.990, Y  +664.041, Z    +0.000, E1    +9.423, E3 +154999.213}
SPL {X  -159.990, Y  +660.147, Z    +0.000, E1   +17.275, E3 +154999.451}
SPL {X  -159.990, Y  +656.649, Z    +0.000, E1   +24.355, E3 +154999.757}
SPL {X  -159.990, Y  +650.462, Z    +0.000, E1   +35.240, E3 +155000.574}
SPL {X  -159.990, Y  +636.155, Z    +0.000, E1   +51.890, E3 +155003.472}
SPL {X  -159.990, Y  +583.574, Z    +0.000, E1   +66.740, E3 +155023.268}
SPL {X  -159.990, Y  +451.342, Z    +0.000, E1   +68.591, E3 +155108.960}
ENDSPLINE

SPLINE
SPL {X  -159.990, Y  +495.016, Z    +0.000, E1   +61.398, E3 +155122.924}
ENDSPLINE

SPLINE
SPL {X  -159.990, Y  +473.575, Z    +0.000, E1   +62.704, E3 +155137.659}
SPL {X  -159.990, Y  +455.620, Z    +0.000, E1   +63.615, E3 +155150.277}
SPL {X  -159.990, Y  +433.781, Z    +0.000, E1   +64.535, E3 +155165.944}
SPL {X  -159.990, Y  +407.091, Z    +0.000, E1   +65.705, E3 +155183.148}
SPL {X  -159.990, Y  +383.383, Z    +0.000, E1   +66.590, E3 +155198.282}
SPL {X  -158.268, Y  +359.089, Z    +0.000, E1   +67.514, E3 +155212.483}
SPL {X  -153.587, Y  +337.689, Z    +0.000, E1   +68.173, E3 +155225.217}
SPL {X  -150.185, Y  +327.353, Z    +0.000, E1   +67.790, E3 +155236.449}
SPL {X  -147.824, Y  +321.305, Z    +0.000, E1   +67.459, E3 +155243.713}
SPL {X  -144.736, Y  +314.321, Z    +0.000, E1   +67.058, E3 +155252.309}
SPL {X  -140.646, Y  +306.241, Z    +0.000, E1   +66.458, E3 +155262.688}
SPL {X  -137.570, Y  +300.823, Z    +0.000, E1   +65.968, E3 +155269.879}
SPL {X  -133.815, Y  +294.806, Z    +0.000, E1   +65.413, E3 +155277.933}
SPL {X  -130.038, Y  +289.296, Z    +0.000, E1   +64.749, E3 +155285.524}
SPL {X  -127.114, Y  +285.347, Z    +0.000, E1   +64.250, E3 +155290.947}
SPL {X   -96.237, Y  +254.690, Z    +0.000, E1   +52.223, E3 +155434.335}
ENDSPLINE

SPLINE
SPL {X  -139.640, Y  +304.414, Z    +0.000, E1   +43.367, E3 +155554.696}
SPL {X  -154.086, Y  +339.440, Z    +0.000, E1   +30.439, E3 +155570.253}
SPL {X  -158.589, Y  +361.372, Z    +0.000, E1   +17.765, E3 +155574.633}
SPL {X  -159.702, Y  +372.901, Z    +0.000, E1    +9.563, E3 +155575.865}
SPL {X  -159.980, Y  +380.731, Z    +0.000, E1    +3.359, E3 +155576.263}
SPL {X  -159.990, Y  +384.708, Z    +0.000, E1    -0.166, E3 +155576.322}
SPL {X  -159.990, Y  +387.941, Z    +0.000, E1    -5.453, E3 +155576.390}
SPL {X  -159.990, Y  +392.683, Z    +0.000, E1   -14.335, E3 +155576.647}
SPL {X  -159.990, Y  +399.462, Z    +0.000, E1   -27.551, E3 +155577.333}
SPL {X  -159.990, Y  +406.707, Z    +0.000, E1   -39.277, E3 +155578.489}
SPL {X  -159.990, Y  +418.467, Z    +0.000, E1   -51.591, E3 +155581.095}
SPL {X  -159.990, Y  +469.047, Z    +0.000, E1   -66.225, E3 +155600.172}
SPL {X  -159.990, Y  +610.501, Z    +0.000, E1   -69.067, E3 +155687.776}
SPL {X  -159.990, Y  +623.913, Z    +0.000, E1   -69.046, E3 +155698.724}
SPL {X  -159.990, Y  +635.131, Z    +0.000, E1   -69.053, E3 +155707.825}
SPL {X  -159.990, Y  +648.088, Z    +0.000, E1   -69.056, E3 +155718.332}
SPL {X  -159.990, Y  +663.340, Z    +0.000, E1   -69.061, E3 +155730.718}
SPL {X  -159.706, Y  +681.022, Z    +0.000, E1   -69.040, E3 +155745.351}
SPL {X  -158.115, Y  +695.924, Z    +0.000, E1   -68.836, E3 +155759.152}
SPL {X  -156.463, Y  +704.909, Z    +0.000, E1   -68.615, E3 +155768.209}
SPL {X  -154.598, Y  +712.687, Z    +0.000, E1   -68.393, E3 +155776.424}
SPL {X  -151.859, Y  +721.854, Z    +0.000, E1   -68.046, E3 +155786.643}
SPL {X  -148.628, Y  +730.715, Z    +0.000, E1   -67.614, E3 +155797.052}
SPL {X  -145.416, Y  +738.215, Z    +0.000, E1   -67.166, E3 +155806.260}
SPL {X  -142.090, Y  +745.034, Z    +0.000, E1   -66.692, E3 +155814.916}
SPL {X  -138.343, Y  +751.861, Z    +0.000, E1   -66.137, E3 +155823.843}
SPL {X  -133.893, Y  +759.076, Z    +0.000, E1   -65.453, E3 +155833.519}
SPL {X  -129.174, Y  +765.898, Z    +0.000, E1   -64.663, E3 +155842.848}
SPL {X  -126.079, Y  +769.993, Z    +0.000, E1   -64.086, E3 +155848.512}
SPL {X   -94.830, Y  +800.357, Z    +0.000, E1   -53.815, E3 +155960.645}
ENDSPLINE

SPLINE
SPL {X  -133.930, Y  +759.019, Z    +0.000, E1   -46.142, E3 +156108.028}
SPL {X  -149.331, Y  +728.920, Z    +0.000, E1   -37.154, E3 +156125.199}
SPL {X  -155.856, Y  +707.636, Z    +0.000, E1   -27.210, E3 +156131.202}
SPL {X  -158.677, Y  +691.955, Z    +0.000, E1   -17.570, E3 +156133.908}
SPL {X  -159.802, Y  +679.261, Z    +0.000, E1    -8.330, E3 +156135.104}
SPL {X  -159.990, Y  +671.355, Z    +0.000, E1    -1.732, E3 +156135.414}
SPL {X  -159.990, Y  +669.500, Z    +0.000, E1    +0.000, E3 +156135.431}
SPL {X  -159.990, Y  +667.882, Z    +0.000, E1    +2.380, E3 +156135.451}
SPL {X  -159.990, Y  +664.041, Z    +0.000, E1    +9.423, E3 +156135.577}
SPL {X  -159.990, Y  +658.864, Z    +0.000, E1   +19.708, E3 +156135.927}
SPL {X  -159.990, Y  +650.462, Z    +0.000, E1   +35.240, E3 +156136.938}
SPL {X  -159.990, Y  +636.155, Z    +0.000, E1   +51.890, E3 +156139.835}
SPL {X  -159.990, Y  +583.574, Z    +0.000, E1   +66.740, E3 +156159.631}
SPL {X  -159.990, Y  +451.342, Z    +0.000, E1   +68.591, E3 +156245.323}
ENDSPLINE

SPLINE
SPL {X  -159.990, Y  +495.016, Z    +0.000, E1   +61.398, E3 +156259.288}
ENDSPLINE

SPLINE
SPL {X  -159.990, Y  +473.575, Z    +0.000, E1   +62.704, E3 +156274.022}
SPL {X  -159.990, Y  +455.620, Z    +0.000, E1   +63.615, E3 +156286.641}
SPL {X  -159.990, Y  +433.781, Z    +0.000, E1   +64.535, E3 +156302.308}
SPL {X  -159.990, Y  +407.091, Z    +0.000, E1   +65.705, E3 +156319.512}
SPL {X  -159.990, Y  +383.383, Z    +0.000, E1   +66.590, E3 +156334.646}
SPL {X  -158.268, Y  +359.089, Z    +0.000, E1   +67.514, E3 +156348.847}
SPL {X  -153.587, Y  +337.689, Z    +0.000, E1   +68.173, E3 +156361.581}
SPL {X  -150.185, Y  +327.353, Z    +0.000, E1   +67.790, E3 +156372.813}
SPL {X  -147.050, Y  +319.468, Z    +0.000, E1   +67.370, E3 +156382.294}
SPL {X  -142.939, Y  +310.631, Z    +0.000, E1   +66.808, E3 +156393.348}
SPL {X  -138.502, Y  +302.413, Z    +0.000, E1   +66.138, E3 +156404.090}
SPL {X  -135.296, Y  +297.108, Z    +0.000, E1   +65.610, E3 +156411.230}
SPL {X  -132.805, Y  +293.283, Z    +0.000, E1   +65.214, E3 +156416.413}
SPL {X  -130.038, Y  +289.296, Z    +0.000, E1   +64.749, E3 +156421.888}
SPL {X  -127.114, Y  +285.347, Z    +0.000, E1   +64.250, E3 +156427.311}
SPL {X   -96.237, Y  +254.690, Z    +0.000, E1   +52.223, E3 +156570.699}
ENDSPLINE

SPLINE
SPL {X  -139.640, Y  +304.414, Z    +0.000, E1   +43.367, E3 +156691.060}
SPL {X  -151.122, Y  +329.974, Z    +0.000, E1   +34.701, E3 +156703.852}
SPL {X  -155.699, Y  +345.695, Z    +0.000, E1   +27.167, E3 +156708.232}
SPL {X  -158.589, Y  +361.372, Z    +0.000, E1   +17.765, E3 +156710.997}
SPL {X  -159.702, Y  +372.901, Z    +0.000, E1    +9.563, E3 +156712.229}
SPL {X  -159.980, Y  +380.731, Z    +0.000, E1    +3.359, E3 +156712.627}
SPL {X  -159.990, Y  +384.465, Z    +0.000, E1    +0.049, E3 +156712.684}
SPL {X  -159.990, Y  +386.161, Z    +0.000, E1    -2.359, E3 +156712.706}
SPL {X  -159.990, Y  +391.786, Z    +0.000, E1   -12.382, E3 +156712.957}
SPL {X  -159.990, Y  +399.462, Z    +0.000, E1   -27.551, E3 +156713.697}
SPL {X  -159.990, Y  +406.707, Z    +0.000, E1   -39.277, E3 +156714.853}
SPL {X  -159.990, Y  +418.467, Z    +0.000, E1   -51.591, E3 +156717.458}
SPL {X  -159.990, Y  +469.047, Z    +0.000, E1   -66.225, E3 +156736.535}
SPL {X  -159.990, Y  +610.501, Z    +0.000, E1   -69.067, E3 +156824.139}
SPL {X  -159.990, Y  +623.913, Z    +0.000, E1   -69.046, E3 +156835.088}
SPL {X  -159.990, Y  +635.131, Z    +0.000, E1   -69.053, E3 +156844.189}
SPL {X  -159.990, Y  +652.219, Z    +0.000, E1   -69.078, E3 +156858.004}
SPL {X  -159.990, Y  +671.254, Z    +0.000, E1   -69.063, E3 +156873.505}
SPL {X  -159.471, Y  +684.377, Z    +0.000, E1   -68.989, E3 +156884.732}
SPL {X  -158.115, Y  +695.924, Z    +0.000, E1   -68.836, E3 +156895.516}
SPL {X  -156.463, Y  +704.909, Z    +0.000, E1   -68.615, E3 +156904.573}
SPL {X  -153.837, Y  +715.444, Z    +0.000, E1   -68.325, E3 +156915.750}
SPL {X  -151.088, Y  +724.124, Z    +0.000, E1   -67.925, E3 +156925.661}
SPL {X  -148.628, Y  +730.715, Z    +0.000, E1   -67.614, E3 +156933.415}
SPL {X  -145.416, Y  +738.215, Z    +0.000, E1   -67.166, E3 +156942.624}
SPL {X  -142.090, Y  +745.034, Z    +0.000, E1   -66.692, E3 +156951.279}
SPL {X  -138.343, Y  +751.861, Z    +0.000, E1   -66.137, E3 +156960.206}
SPL {X  -133.893, Y  +759.076, Z    +0.000, E1   -65.453, E3 +156969.882}
SPL {X  -130.341, Y  +764.280, Z    +0.000, E1   -64.831, E3 +156977.021}
SPL {X  -127.405, Y  +768.272, Z    +0.000, E1   -64.349, E3 +156982.476}
SPL {X   -94.830, Y  +800.357, Z    +0.000, E1   -53.815, E3 +157097.008}
ENDSPLINE

SPLINE
SPL {X  -133.930, Y  +759.019, Z    +0.000, E1   -46.142, E3 +157244.392}
SPL {X  -149.331, Y  +728.920, Z    +0.000, E1   -37.154, E3 +157261.562}
SPL {X  -155.856, Y  +707.636, Z    +0.000, E1   -27.210, E3 +157267.566}
SPL {X  -158.677, Y  +691.955, Z    +0.000, E1   -17.570, E3 +157270.271}
SPL {X  -159.802, Y  +679.261, Z    +0.000, E1    -8.330, E3 +157271.468}
SPL {X  -159.990, Y  +671.355, Z    +0.000, E1    -1.732, E3 +157271.778}
SPL {X  -159.990, Y  +669.259, Z    +0.000, E1    +0.225, E3 +157271.797}
SPL {X  -159.990, Y  +665.054, Z    +0.000, E1    +7.292, E3 +157271.902}
SPL {X  -159.990, Y  +658.864, Z    +0.000, E1   +19.708, E3 +157272.290}
SPL {X  -159.990, Y  +650.462, Z    +0.000, E1   +35.240, E3 +157273.301}
SPL {X  -159.990, Y  +636.155, Z    +0.000, E1   +51.890, E3 +157276.199}
SPL {X  -159.990, Y  +583.574, Z    +0.000, E1   +66.740, E3 +157295.995}
SPL {X  -159.990, Y  +451.342, Z    +0.000, E1   +68.591, E3 +157381.687}
ENDSPLINE

SPLINE
SPL {X  -159.990, Y  +495.016, Z    +0.000, E1   +61.398, E3 +157395.651}
ENDSPLINE

SPLINE
SPL {X  -159.990, Y  +473.575, Z    +0.000, E1   +62.704, E3 +157410.386}
SPL {X  -159.990, Y  +455.620, Z    +0.000, E1   +63.615, E3 +157423.004}
SPL {X  -159.990, Y  +433.781, Z    +0.000, E1   +64.535, E3 +157438.672}
SPL {X  -159.990, Y  +414.623, Z    +0.000, E1   +65.374, E3 +157451.092}
SPL {X  -159.990, Y  +395.826, Z    +0.000, E1   +66.138, E3 +157463.106}
SPL {X  -159.536, Y  +370.459, Z    +0.000, E1   +67.052, E3 +157478.999}
SPL {X  -155.924, Y  +346.662, Z    +0.000, E1   +68.026, E3 +157491.624}
SPL {X  -152.751, Y  +334.918, Z    +0.000, E1   +68.124, E3 +157500.454}
SPL {X  -150.185, Y  +327.353, Z    +0.000, E1   +67.790, E3 +157509.177}
SPL {X  -147.824, Y  +321.305, Z    +0.000, E1   +67.459, E3 +157516.440}
SPL {X  -144.736, Y  +314.321, Z    +0.000, E1   +67.058, E3 +157525.036}
SPL {X  -140.646, Y  +306.241, Z    +0.000, E1   +66.458, E3 +157535.415}
SPL {X  -137.570, Y  +300.823, Z    +0.000, E1   +65.968, E3 +157542.607}
SPL {X  -133.815, Y  +294.806, Z    +0.000, E1   +65.413, E3 +157550.660}
SPL {X  -130.038, Y  +289.296, Z    +0.000, E1   +64.749, E3 +157558.251}
SPL {X  -127.114, Y  +285.347, Z    +0.000, E1   +64.250, E3 +157563.674}
SPL {X   -96.237, Y  +254.690, Z    +0.000, E1   +52.223, E3 +157707.062}
ENDSPLINE

SPLINE
SPL {X  -139.640, Y  +304.414, Z    +0.000, E1   +43.367, E3 +157827.423}
SPL {X  -154.086, Y  +339.440, Z    +0.000, E1   +30.439, E3 +157842.981}
SPL {X  -158.589, Y  +361.372, Z    +0.000, E1   +17.765, E3 +157847.360}
SPL {X  -159.702, Y  +372.901, Z    +0.000, E1    +9.563, E3 +157848.592}
SPL {X  -159.980, Y  +380.731, Z    +0.000, E1    +3.359, E3 +157848.990}
SPL {X  -159.990, Y  +384.465, Z    +0.000, E1    +0.049, E3 +157849.048}
SPL {X  -159.990, Y  +386.161, Z    +0.000, E1    -2.359, E3 +157849.070}
SPL {X  -159.990, Y  +391.786, Z    +0.000, E1   -12.382, E3 +157849.321}
SPL {X  -159.990, Y  +399.462, Z    +0.000, E1   -27.551, E3 +157850.061}
SPL {X  -159.990, Y  +406.707, Z    +0.000, E1   -39.277, E3 +157851.216}
SPL {X  -159.990, Y  +418.467, Z    +0.000, E1   -51.591, E3 +157853.822}
SPL {X  -159.990, Y  +469.047, Z    +0.000, E1   -66.225, E3 +157872.899}
SPL {X  -159.990, Y  +610.501, Z    +0.000, E1   -69.067, E3 +157960.503}
SPL {X  -159.990, Y  +630.690, Z    +0.000, E1   -69.080, E3 +157976.883}
SPL {X  -159.990, Y  +648.088, Z    +0.000, E1   -69.056, E3 +157991.060}
SPL {X  -159.990, Y  +663.340, Z    +0.000, E1   -69.061, E3 +158003.446}
SPL {X  -159.706, Y  +681.022, Z    +0.000, E1   -69.040, E3 +158018.078}
SPL {X  -158.115, Y  +695.924, Z    +0.000, E1   -68.836, E3 +158031.879}
SPL {X  -156.463, Y  +704.909, Z    +0.000, E1   -68.615, E3 +158040.937}
SPL {X  -153.837, Y  +715.444, Z    +0.000, E1   -68.325, E3 +158052.114}
SPL {X  -151.088, Y  +724.124, Z    +0.000, E1   -67.925, E3 +158062.024}
SPL {X  -148.628, Y  +730.715, Z    +0.000, E1   -67.614, E3 +158069.779}
SPL {X  -145.416, Y  +738.215, Z    +0.000, E1   -67.166, E3 +158078.988}
SPL {X  -141.128, Y  +746.863, Z    +0.000, E1   -66.582, E3 +158089.964}
SPL {X  -137.485, Y  +753.321, Z    +0.000, E1   -65.984, E3 +158098.541}
SPL {X  -134.819, Y  +757.643, Z    +0.000, E1   -65.575, E3 +158104.336}
SPL {X  -131.187, Y  +763.079, Z    +0.000, E1   -64.994, E3 +158111.719}
SPL {X  -127.405, Y  +768.272, Z    +0.000, E1   -64.349, E3 +158118.840}
SPL {X   -94.830, Y  +800.357, Z    +0.000, E1   -53.815, E3 +158233.372}
ENDSPLINE

SPLINE
SPL {X  -133.930, Y  +759.019, Z    +0.000, E1   -46.142, E3 +158380.755}
SPL {X  -149.331, Y  +728.920, Z    +0.000, E1   -37.154, E3 +158397.926}
SPL {X  -155.856, Y  +707.636, Z    +0.000, E1   -27.210, E3 +158403.929}
SPL {X  -159.260, Y  +686.764, Z    +0.000, E1   -14.026, E3 +158407.204}
SPL {X  -159.985, Y  +672.780, Z    +0.000, E1    -3.059, E3 +158408.105}
SPL {X  -159.990, Y  +669.259, Z    +0.000, E1    +0.225, E3 +158408.160}
SPL {X  -159.990, Y  +665.054, Z    +0.000, E1    +7.292, E3 +158408.265}
SPL {X  -159.990, Y  +658.864, Z    +0.000, E1   +19.708, E3 +158408.654}
SPL {X  -159.990, Y  +650.462, Z    +0.000, E1   +35.240, E3 +158409.665}
SPL {X  -159.990, Y  +636.155, Z    +0.000, E1   +51.890, E3 +158412.563}
SPL {X  -159.990, Y  +583.574, Z    +0.000, E1   +66.740, E3 +158432.359}
SPL {X  -159.990, Y  +451.342, Z    +0.000, E1   +68.591, E3 +158518.051}
ENDSPLINE

SPLINE
SPL {X  -159.990, Y  +495.016, Z    +0.000, E1   +61.398, E3 +158532.015}
ENDSPLINE

SPLINE
SPL {X  -159.990, Y  +473.575, Z    +0.000, E1   +62.704, E3 +158546.750}
SPL {X  -159.990, Y  +455.620, Z    +0.000, E1   +63.615, E3 +158559.368}
SPL {X  -159.990, Y  +439.579, Z    +0.000, E1   +64.263, E3 +158571.103}
SPL {X  -159.990, Y  +420.812, Z    +0.000, E1   +65.111, E3 +158583.535}
SPL {X  -159.990, Y  +395.826, Z    +0.000, E1   +66.138, E3 +158599.470}
SPL {X  -159.536, Y  +370.459, Z    +0.000, E1   +67.052, E3 +158615.363}
SPL {X  -155.924, Y  +346.662, Z    +0.000, E1   +68.026, E3 +158627.988}
SPL {X  -152.751, Y  +334.918, Z    +0.000, E1   +68.124, E3 +158636.818}
SPL {X  -150.185, Y  +327.353, Z    +0.000, E1   +67.790, E3 +158645.540}
SPL {X  -147.050, Y  +319.468, Z    +0.000, E1   +67.370, E3 +158655.021}
SPL {X  -143.990, Y  +312.760, Z    +0.000, E1   +66.929, E3 +158663.410}
SPL {X  -140.646, Y  +306.241, Z    +0.000, E1   +66.458, E3 +158671.779}
SPL {X  -136.388, Y  +298.863, Z    +0.000, E1   +65.814, E3 +158681.551}
SPL {X  -132.805, Y  +293.283, Z    +0.000, E1   +65.214, E3 +158689.141}
SPL {X  -130.038, Y  +289.296, Z    +0.000, E1   +64.749, E3 +158694.615}
SPL {X  -127.114, Y  +285.347, Z    +0.000, E1   +64.250, E3 +158700.038}
SPL {X   -96.237, Y  +254.690, Z    +0.000, E1   +52.223, E3 +158843.426}
ENDSPLINE

SPLINE
SPL {X  -139.640, Y  +304.414, Z    +0.000, E1   +43.367, E3 +158963.787}
SPL {X  -154.086, Y  +339.440, Z    +0.000, E1   +30.439, E3 +158979.344}
SPL {X  -158.589, Y  +361.372, Z    +0.000, E1   +17.765, E3 +158983.724}
SPL {X  -159.702, Y  +372.901, Z    +0.000, E1    +9.563, E3 +158984.956}
SPL {X  -159.980, Y  +380.731, Z    +0.000, E1    +3.359, E3 +158985.354}
SPL {X  -159.990, Y  +384.465, Z    +0.000, E1    +0.049, E3 +158985.411}
SPL {X  -159.990, Y  +386.161, Z    +0.000, E1    -2.359, E3 +158985.434}
SPL {X  -159.990, Y  +390.716, Z    +0.000, E1   -10.524, E3 +158985.609}
SPL {X  -159.990, Y  +397.792, Z    +0.000, E1   -24.215, E3 +158986.239}
SPL {X  -159.990, Y  +406.707, Z    +0.000, E1   -39.277, E3 +158987.580}
SPL {X  -159.990, Y  +418.467, Z    +0.000, E1   -51.591, E3 +158990.185}
SPL {X  -159.990, Y  +469.047, Z    +0.000, E1   -66.225, E3 +159009.263}
SPL {X  -159.990, Y  +610.501, Z    +0.000, E1   -69.067, E3 +159096.867}
SPL {X  -159.990, Y  +630.690, Z    +0.000, E1   -69.080, E3 +159113.247}
SPL {X  -159.990, Y  +652.219, Z    +0.000, E1   -69.078, E3 +159130.731}
SPL {X  -159.990, Y  +671.254, Z    +0.000, E1   -69.063, E3 +159146.232}
SPL {X  -159.172, Y  +687.655, Z    +0.000, E1   -68.973, E3 +159160.391}
SPL {X  -157.106, Y  +701.739, Z    +0.000, E1   -68.720, E3 +159174.000}
SPL {X  -153.837, Y  +715.444, Z    +0.000, E1   -68.325, E3 +159188.478}
SPL {X  -151.088, Y  +724.124, Z    +0.000, E1   -67.925, E3 +159198.388}
SPL {X  -148.628, Y  +730.715, Z    +0.000, E1   -67.614, E3 +159206.143}
SPL {X  -145.416, Y  +738.215, Z    +0.000, E1   -67.166, E3 +159215.351}
SPL {X  -142.090, Y  +745.034, Z    +0.000, E1   -66.692, E3 +159224.007}
SPL {X  -138.343, Y  +751.861, Z    +0.000, E1   -66.137, E3 +159232.934}
SPL {X  -133.893, Y  +759.076, Z    +0.000, E1   -65.453, E3 +159242.610}
SPL {X  -130.341, Y  +764.280, Z    +0.000, E1   -64.831, E3 +159249.748}
SPL {X  -127.405, Y  +768.272, Z    +0.000, E1   -64.349, E3 +159255.203}
SPL {X   -94.830, Y  +800.357, Z    +0.000, E1   -53.815, E3 +159369.736}
ENDSPLINE

SPLINE
SPL {X  -133.930, Y  +759.019, Z    +0.000, E1   -46.142, E3 +159517.119}
SPL {X  -149.331, Y  +728.920, Z    +0.000, E1   -37.154, E3 +159534.290}
SPL {X  -155.856, Y  +707.636, Z    +0.000, E1   -27.210, E3 +159540.293}
SPL {X  -158.677, Y  +691.955, Z    +0.000, E1   -17.570, E3 +159542.999}
SPL {X  -159.802, Y  +679.261, Z    +0.000, E1    -8.330, E3 +159544.195}
SPL {X  -159.990, Y  +669.483, Z    +0.000, E1    -0.154, E3 +159544.522}
SPL {X  -159.990, Y  +665.054, Z    +0.000, E1    +7.292, E3 +159544.629}
SPL {X  -159.990, Y  +660.147, Z    +0.000, E1   +17.275, E3 +159544.905}
SPL {X  -159.990, Y  +656.649, Z    +0.000, E1   +24.355, E3 +159545.212}
SPL {X  -159.990, Y  +650.462, Z    +0.000, E1   +35.240, E3 +159546.029}
SPL {X  -159.990, Y  +636.155, Z    +0.000, E1   +51.890, E3 +159548.926}
SPL {X  -159.990, Y  +583.574, Z    +0.000, E1   +66.740, E3 +159568.722}
SPL {X  -159.990, Y  +451.342, Z    +0.000, E1   +68.591, E3 +159654.414}
ENDSPLINE

SPLINE
SPL {X  -159.990, Y  +495.016, Z    +0.000, E1   +61.398, E3 +159668.379}
ENDSPLINE

SPLINE
SPL {X  -159.990, Y  +473.575, Z    +0.000, E1   +62.704, E3 +159683.113}
SPL {X  -159.990, Y  +455.620, Z    +0.000, E1   +63.615, E3 +159695.731}
SPL {X  -159.990, Y  +433.781, Z    +0.000, E1   +64.535, E3 +159711.399}
SPL {X  -159.990, Y  +407.091, Z    +0.000, E1   +65.705, E3 +159728.602}
SPL {X  -159.990, Y  +383.383, Z    +0.000, E1   +66.590, E3 +159743.737}
SPL {X  -158.268, Y  +359.089, Z    +0.000, E1   +67.514, E3 +159757.938}
SPL {X  -153.587, Y  +337.689, Z    +0.000, E1   +68.173, E3 +159770.672}
SPL {X  -150.185, Y  +327.353, Z    +0.000, E1   +67.790, E3 +159781.904}
SPL {X  -147.050, Y  +319.468, Z    +0.000, E1   +67.370, E3 +159791.385}
SPL {X  -142.939, Y  +310.631, Z    +0.000, E1   +66.808, E3 +159802.438}
SPL {X  -138.502, Y  +302.413, Z    +0.000, E1   +66.138, E3 +159813.181}
SPL {X  -133.815, Y  +294.806, Z    +0.000, E1   +65.413, E3 +159823.387}
SPL {X  -130.038, Y  +289.296, Z    +0.000, E1   +64.749, E3 +159830.979}
SPL {X  -127.114, Y  +285.347, Z    +0.000, E1   +64.250, E3 +159836.402}
SPL {X   -96.237, Y  +254.690, Z    +0.000, E1   +52.223, E3 +159979.790}
ENDSPLINE

SPLINE
SPL {X  -139.640, Y  +304.414, Z    +0.000, E1   +43.367, E3 +160100.151}
SPL {X  -154.086, Y  +339.440, Z    +0.000, E1   +30.439, E3 +160115.708}
SPL {X  -158.589, Y  +361.372, Z    +0.000, E1   +17.765, E3 +160120.088}
SPL {X  -159.702, Y  +372.901, Z    +0.000, E1    +9.563, E3 +160121.320}
SPL {X  -159.980, Y  +380.731, Z    +0.000, E1    +3.359, E3 +160121.717}
SPL {X  -159.990, Y  +384.465, Z    +0.000, E1    +0.049, E3 +160121.775}
SPL {X  -159.990, Y  +386.161, Z    +0.000, E1    -2.359, E3 +160121.797}
SPL {X  -159.990, Y  +390.716, Z    +0.000, E1   -10.524, E3 +160121.973}
SPL {X  -159.990, Y  +397.792, Z    +0.000, E1   -24.215, E3 +160122.602}
SPL {X  -159.990, Y  +406.707, Z    +0.000, E1   -39.277, E3 +160123.943}
SPL {X  -159.990, Y  +418.467, Z    +0.000, E1   -51.591, E3 +160126.549}
SPL {X  -159.990, Y  +469.047, Z    +0.000, E1   -66.225, E3 +160145.626}
SPL {X  -159.990, Y  +610.501, Z    +0.000, E1   -69.067, E3 +160233.230}
SPL {X  -159.990, Y  +630.690, Z    +0.000, E1   -69.080, E3 +160249.611}
SPL {X  -159.990, Y  +652.219, Z    +0.000, E1   -69.078, E3 +160267.095}
SPL {X  -159.990, Y  +671.254, Z    +0.000, E1   -69.063, E3 +160282.596}
SPL {X  -159.172, Y  +687.655, Z    +0.000, E1   -68.973, E3 +160296.755}
SPL {X  -157.106, Y  +701.739, Z    +0.000, E1   -68.720, E3 +160310.363}
SPL {X  -154.598, Y  +712.687, Z    +0.000, E1   -68.393, E3 +160321.878}
SPL {X  -151.859, Y  +721.854, Z    +0.000, E1   -68.046, E3 +160332.097}
SPL {X  -148.628, Y  +730.715, Z    +0.000, E1   -67.614, E3 +160342.506}
SPL {X  -145.416, Y  +738.215, Z    +0.000, E1   -67.166, E3 +160351.715}
SPL {X  -142.090, Y  +745.034, Z    +0.000, E1   -66.692, E3 +160360.370}
SPL {X  -138.343, Y  +751.861, Z    +0.000, E1   -66.137, E3 +160369.297}
SPL {X  -134.819, Y  +757.643, Z    +0.000, E1   -65.575, E3 +160377.063}
SPL {X  -131.187, Y  +763.079, Z    +0.000, E1   -64.994, E3 +160384.447}
SPL {X  -127.405, Y  +768.272, Z    +0.000, E1   -64.349, E3 +160391.567}
SPL {X   -94.830, Y  +800.357, Z    +0.000, E1   -53.815, E3 +160506.099}
ENDSPLINE

